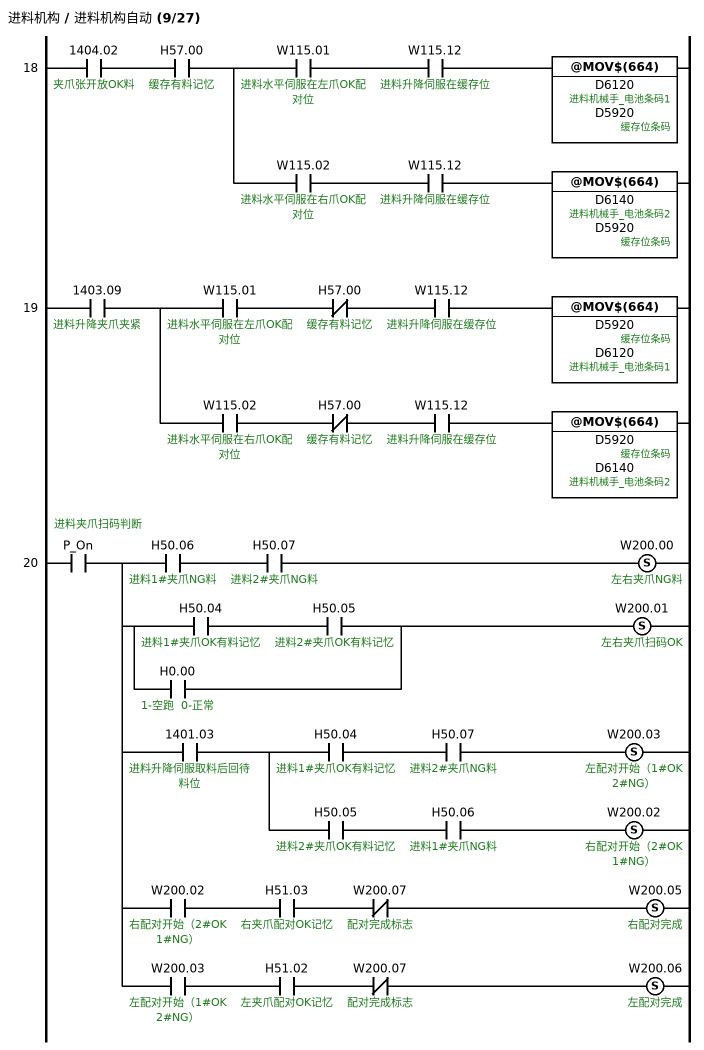
; rung 18
LD 1404.02  ; 夹爪张开放OK料
AND H57.00  ; 缓存有料记忆
OUT TR0
AND W115.01  ; 进料水平伺服在左爪OK配对位
AND W115.12  ; 进料升降伺服在缓存位
@MOV$(664) D6120 D5920  ; 进料机械手_电池条码1, 缓存位条码
LD TR0
AND W115.02  ; 进料水平伺服在右爪OK配对位
AND W115.12  ; 进料升降伺服在缓存位
@MOV$(664) D6140 D5920  ; 进料机械手_电池条码2, 缓存位条码
; rung 19
LD 1403.09  ; 进料升降夹爪夹紧
OUT TR0
AND W115.01  ; 进料水平伺服在左爪OK配对位
ANDNOT H57.00  ; 缓存有料记忆
AND W115.12  ; 进料升降伺服在缓存位
@MOV$(664) D5920 D6120  ; 缓存位条码, 进料机械手_电池条码1
LD TR0
AND W115.02  ; 进料水平伺服在右爪OK配对位
ANDNOT H57.00  ; 缓存有料记忆
AND W115.12  ; 进料升降伺服在缓存位
@MOV$(664) D5920 D6140  ; 缓存位条码, 进料机械手_电池条码2
; rung 20: 进料夹爪扫码判断
LD P_On
OUT TR0
AND H50.06  ; 进料1#夹爪NG料
AND H50.07  ; 进料2#夹爪NG料
SET W200.00  ; 左右夹爪NG料
LD TR0
LD H50.04  ; 进料1#夹爪OK有料记忆
AND H50.05  ; 进料2#夹爪OK有料记忆
OR H0.00  ; 1-空跑  0-正常
ANDLD
SET W200.01  ; 左右夹爪扫码OK
LD TR0
AND 1401.03  ; 进料升降伺服取料后回待料位
OUT TR1
AND H50.04  ; 进料1#夹爪OK有料记忆
AND H50.07  ; 进料2#夹爪NG料
SET W200.03  ; 左配对开始（1#OK 2#NG）
LD TR1
AND H50.05  ; 进料2#夹爪OK有料记忆
AND H50.06  ; 进料1#夹爪NG料
SET W200.02  ; 右配对开始（2#OK 1#NG）
LD TR0
AND W200.02  ; 右配对开始（2#OK 1#NG）
AND H51.03  ; 右夹爪配对OK记忆
ANDNOT W200.07  ; 配对完成标志
SET W200.05  ; 右配对完成
LD TR0
AND W200.03  ; 左配对开始（1#OK 2#NG）
AND H51.02  ; 左夹爪配对OK记忆
ANDNOT W200.07  ; 配对完成标志
SET W200.06  ; 左配对完成

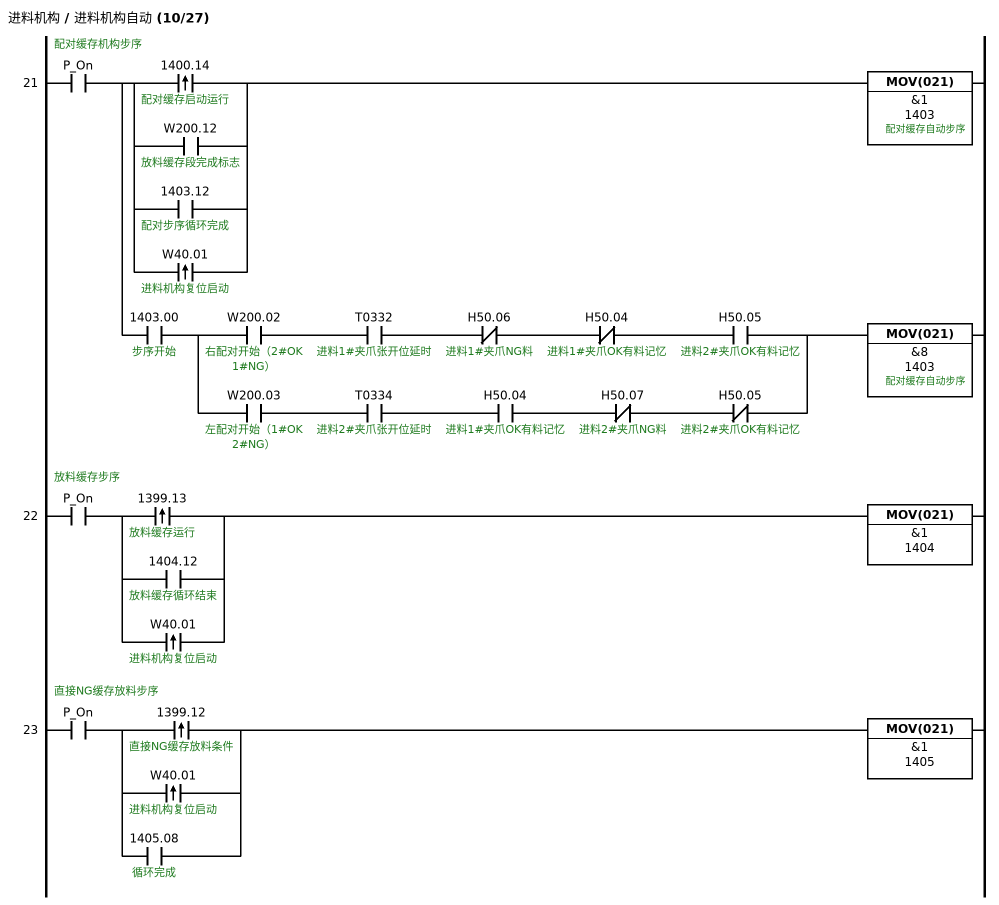
; rung 21: 配对缓存机构步序
LD P_On
OUT TR0
@LD 1400.14  ; 配对缓存启动运行
OR W200.12  ; 放料缓存段完成标志
OR 1403.12  ; 配对步序循环完成
@OR W40.01  ; 进料机构复位启动
ANDLD
MOV(021) &1 1403  ; 配对缓存自动步序
LD TR0
AND 1403.00  ; 步序开始
LD W200.02  ; 右配对开始（2#OK 1#NG）
AND T0332  ; 进料1#夹爪张开位延时
ANDNOT H50.06  ; 进料1#夹爪NG料
ANDNOT H50.04  ; 进料1#夹爪OK有料记忆
AND H50.05  ; 进料2#夹爪OK有料记忆
LD W200.03  ; 左配对开始（1#OK 2#NG）
AND T0334  ; 进料2#夹爪张开位延时
AND H50.04  ; 进料1#夹爪OK有料记忆
ANDNOT H50.07  ; 进料2#夹爪NG料
ANDNOT H50.05  ; 进料2#夹爪OK有料记忆
ORLD
ANDLD
MOV(021) &8 1403  ; 配对缓存自动步序
; rung 22: 放料缓存步序
LD P_On
@LD 1399.13  ; 放料缓存运行
OR 1404.12  ; 放料缓存循环结束
@OR W40.01  ; 进料机构复位启动
ANDLD
MOV(021) &1 1404
; rung 23: 直接NG缓存放料步序
LD P_On
@LD 1399.12  ; 直接NG缓存放料条件
@OR W40.01  ; 进料机构复位启动
OR 1405.08  ; 循环完成
ANDLD
MOV(021) &1 1405

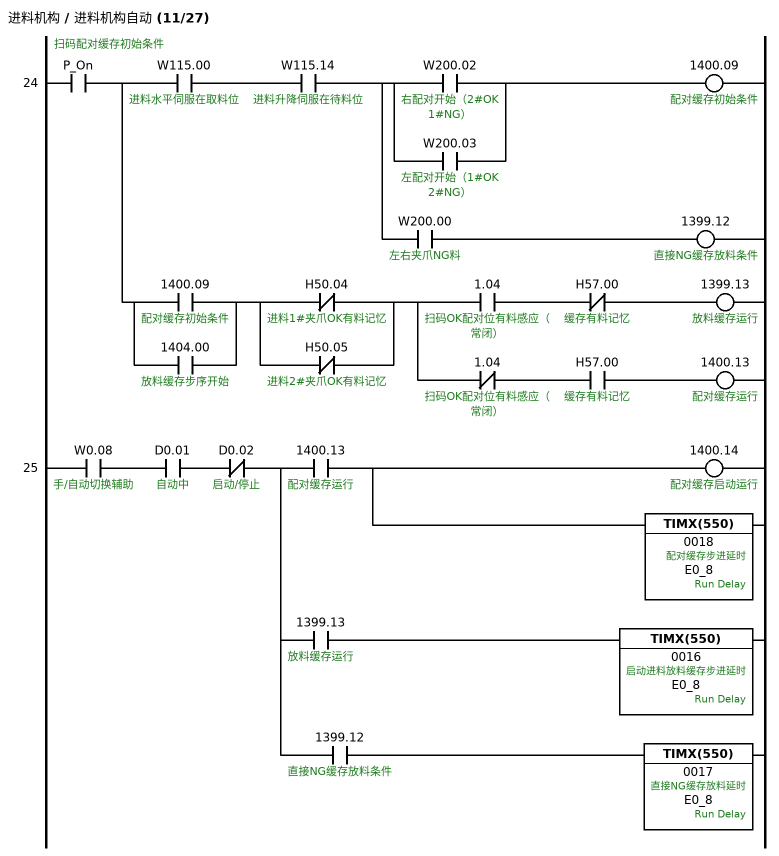
; rung 24: 扫码配对缓存初始条件
LD P_On
OUT TR0
AND W115.00  ; 进料水平伺服在取料位
AND W115.14  ; 进料升降伺服在待料位
OUT TR1
LD W200.02  ; 右配对开始（2#OK 1#NG）
OR W200.03  ; 左配对开始（1#OK 2#NG）
ANDLD
OUT 1400.09  ; 配对缓存初始条件
LD TR1
AND W200.00  ; 左右夹爪NG料
OUT 1399.12  ; 直接NG缓存放料条件
LD TR0
LD 1400.09  ; 配对缓存初始条件
OR 1404.00  ; 放料缓存步序开始
ANDLD
LDNOT H50.04  ; 进料1#夹爪OK有料记忆
ORNOT H50.05  ; 进料2#夹爪OK有料记忆
ANDLD
OUT TR0
AND 1.04  ; 扫码OK配对位有料感应（常闭）
ANDNOT H57.00  ; 缓存有料记忆
OUT 1399.13  ; 放料缓存运行
LD TR0
ANDNOT 1.04  ; 扫码OK配对位有料感应（常闭）
AND H57.00  ; 缓存有料记忆
OUT 1400.13  ; 配对缓存运行
; rung 25
LD W0.08  ; 手/自动切换辅助
AND D0.01  ; 自动中
ANDNOT D0.02  ; 启动/停止
OUT TR0
AND 1400.13  ; 配对缓存运行
OUT 1400.14  ; 配对缓存启动运行
TIMX(550) 0018 E0_8  ; Run Delay, 配对缓存步进延时
LD TR0
AND 1399.13  ; 放料缓存运行
TIMX(550) 0016 E0_8  ; Run Delay, 启动进料放料缓存步进延时
LD TR0
AND 1399.12  ; 直接NG缓存放料条件
TIMX(550) 0017 E0_8  ; Run Delay, 直接NG缓存放料延时

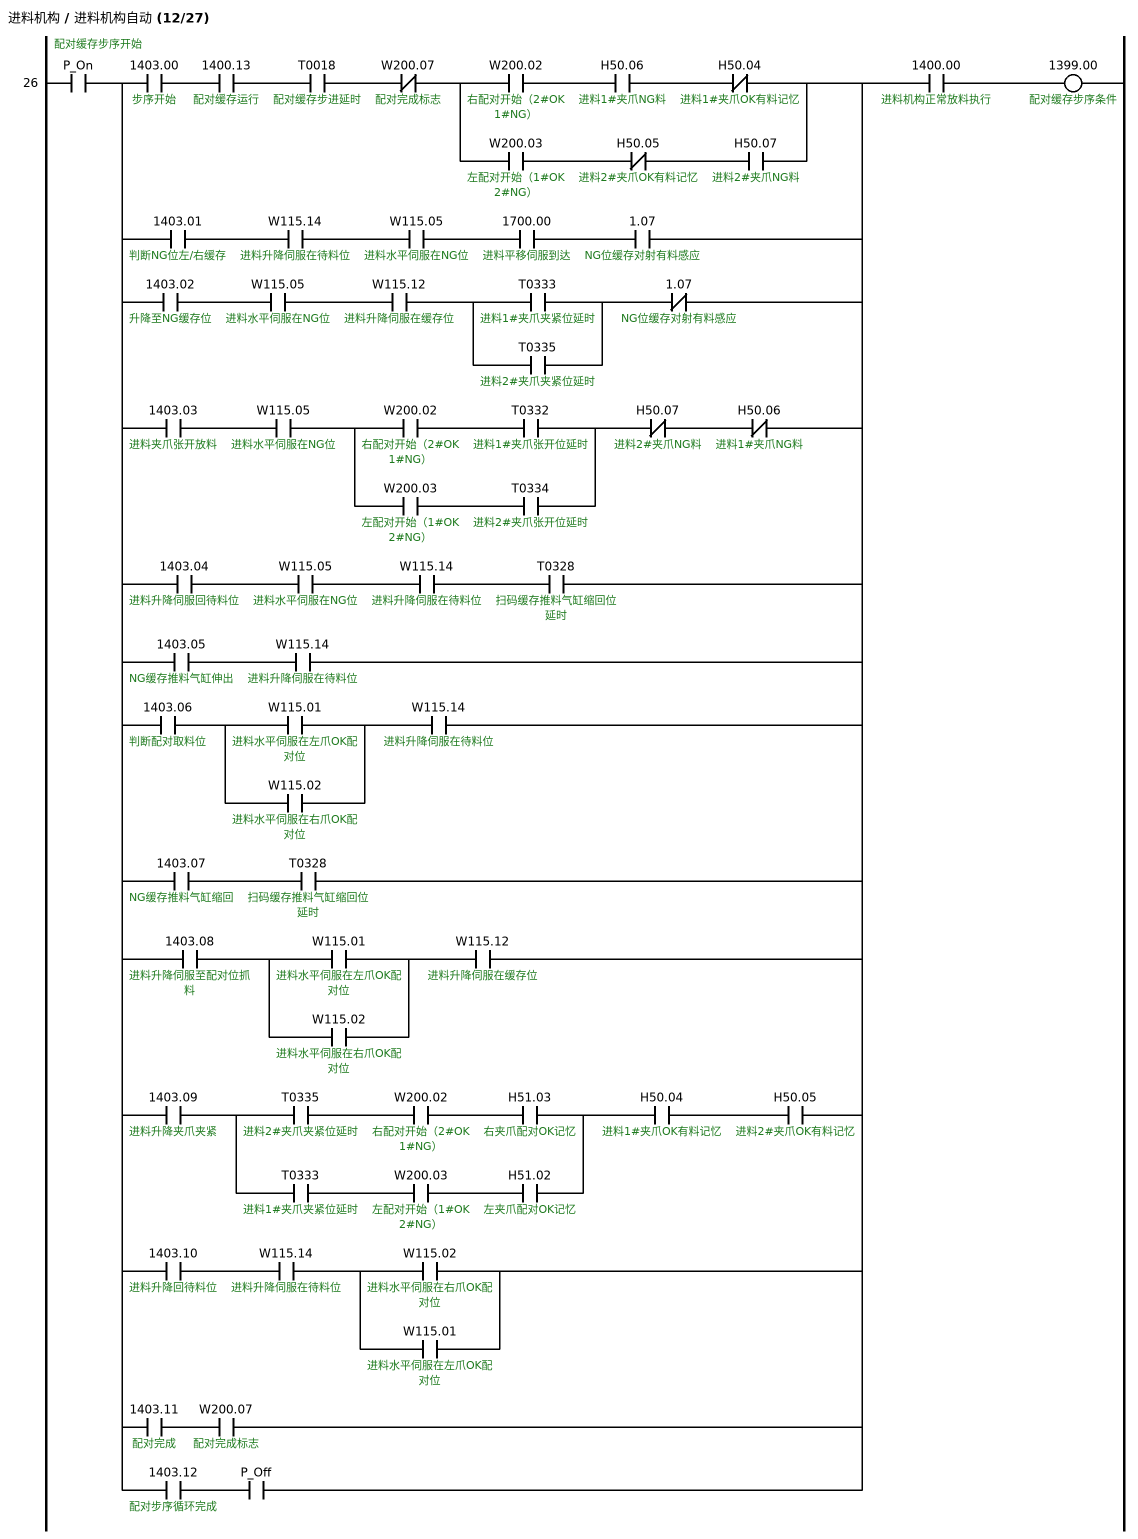
; rung 26: 配对缓存步序开始
LD P_On
LD 1403.00  ; 步序开始
AND 1400.13  ; 配对缓存运行
AND T0018  ; 配对缓存步进延时
ANDNOT W200.07  ; 配对完成标志
LD W200.02  ; 右配对开始（2#OK 1#NG）
AND H50.06  ; 进料1#夹爪NG料
ANDNOT H50.04  ; 进料1#夹爪OK有料记忆
LD W200.03  ; 左配对开始（1#OK 2#NG）
ANDNOT H50.05  ; 进料2#夹爪OK有料记忆
AND H50.07  ; 进料2#夹爪NG料
ORLD
ANDLD
LD 1403.01  ; 判断NG位左/右缓存
AND W115.14  ; 进料升降伺服在待料位
AND W115.05  ; 进料水平伺服在NG位
AND 1700.00  ; 进料平移伺服到达
AND 1.07  ; NG位缓存对射有料感应
ORLD
LD 1403.02  ; 升降至NG缓存位
AND W115.05  ; 进料水平伺服在NG位
AND W115.12  ; 进料升降伺服在缓存位
LD T0333  ; 进料1#夹爪夹紧位延时
OR T0335  ; 进料2#夹爪夹紧位延时
ANDLD
ANDNOT 1.07  ; NG位缓存对射有料感应
ORLD
LD 1403.03  ; 进料夹爪张开放料
AND W115.05  ; 进料水平伺服在NG位
LD W200.02  ; 右配对开始（2#OK 1#NG）
AND T0332  ; 进料1#夹爪张开位延时
LD W200.03  ; 左配对开始（1#OK 2#NG）
AND T0334  ; 进料2#夹爪张开位延时
ORLD
ANDLD
ANDNOT H50.07  ; 进料2#夹爪NG料
ANDNOT H50.06  ; 进料1#夹爪NG料
ORLD
LD 1403.04  ; 进料升降伺服回待料位
AND W115.05  ; 进料水平伺服在NG位
AND W115.14  ; 进料升降伺服在待料位
AND T0328  ; 扫码缓存推料气缸缩回位延时
ORLD
LD 1403.05  ; NG缓存推料气缸伸出
AND W115.14  ; 进料升降伺服在待料位
ORLD
LD 1403.06  ; 判断配对取料位
LD W115.01  ; 进料水平伺服在左爪OK配对位
OR W115.02  ; 进料水平伺服在右爪OK配对位
ANDLD
AND W115.14  ; 进料升降伺服在待料位
ORLD
LD 1403.07  ; NG缓存推料气缸缩回
AND T0328  ; 扫码缓存推料气缸缩回位延时
ORLD
LD 1403.08  ; 进料升降伺服至配对位抓料
LD W115.01  ; 进料水平伺服在左爪OK配对位
OR W115.02  ; 进料水平伺服在右爪OK配对位
ANDLD
AND W115.12  ; 进料升降伺服在缓存位
ORLD
LD 1403.09  ; 进料升降夹爪夹紧
LD T0335  ; 进料2#夹爪夹紧位延时
AND W200.02  ; 右配对开始（2#OK 1#NG）
AND H51.03  ; 右夹爪配对OK记忆
LD T0333  ; 进料1#夹爪夹紧位延时
AND W200.03  ; 左配对开始（1#OK 2#NG）
AND H51.02  ; 左夹爪配对OK记忆
ORLD
ANDLD
AND H50.04  ; 进料1#夹爪OK有料记忆
AND H50.05  ; 进料2#夹爪OK有料记忆
ORLD
LD 1403.10  ; 进料升降回待料位
AND W115.14  ; 进料升降伺服在待料位
LD W115.02  ; 进料水平伺服在右爪OK配对位
OR W115.01  ; 进料水平伺服在左爪OK配对位
ANDLD
ORLD
LD 1403.11  ; 配对完成
AND W200.07  ; 配对完成标志
ORLD
LD 1403.12  ; 配对步序循环完成
AND P_Off
ORLD
ANDLD
AND 1400.00  ; 进料机构正常放料执行
OUT 1399.00  ; 配对缓存步序条件

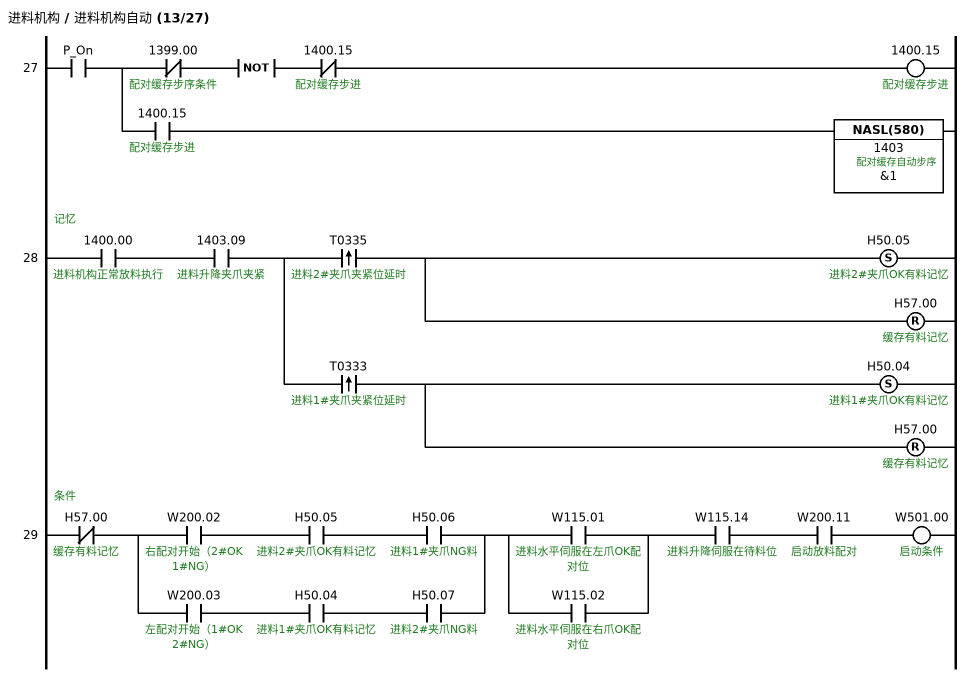
; rung 27
LD P_On
OUT TR0
ANDNOT 1399.00  ; 配对缓存步序条件
NOT(520)
ANDNOT 1400.15  ; 配对缓存步进
OUT 1400.15  ; 配对缓存步进
LD TR0
AND 1400.15  ; 配对缓存步进
NASL(580) 1403 &1  ; 配对缓存自动步序
; rung 28: 记忆
LD 1400.00  ; 进料机构正常放料执行
AND 1403.09  ; 进料升降夹爪夹紧
OUT TR0
@AND T0335  ; 进料2#夹爪夹紧位延时
SET H50.05  ; 进料2#夹爪OK有料记忆
RSET H57.00  ; 缓存有料记忆
LD TR0
@AND T0333  ; 进料1#夹爪夹紧位延时
SET H50.04  ; 进料1#夹爪OK有料记忆
RSET H57.00  ; 缓存有料记忆
; rung 29: 条件
LDNOT H57.00  ; 缓存有料记忆
LD W200.02  ; 右配对开始（2#OK 1#NG）
AND H50.05  ; 进料2#夹爪OK有料记忆
AND H50.06  ; 进料1#夹爪NG料
LD W200.03  ; 左配对开始（1#OK 2#NG）
AND H50.04  ; 进料1#夹爪OK有料记忆
AND H50.07  ; 进料2#夹爪NG料
ORLD
ANDLD
LD W115.01  ; 进料水平伺服在左爪OK配对位
OR W115.02  ; 进料水平伺服在右爪OK配对位
ANDLD
AND W115.14  ; 进料升降伺服在待料位
AND W200.11  ; 启动放料配对
OUT W501.00  ; 启动条件

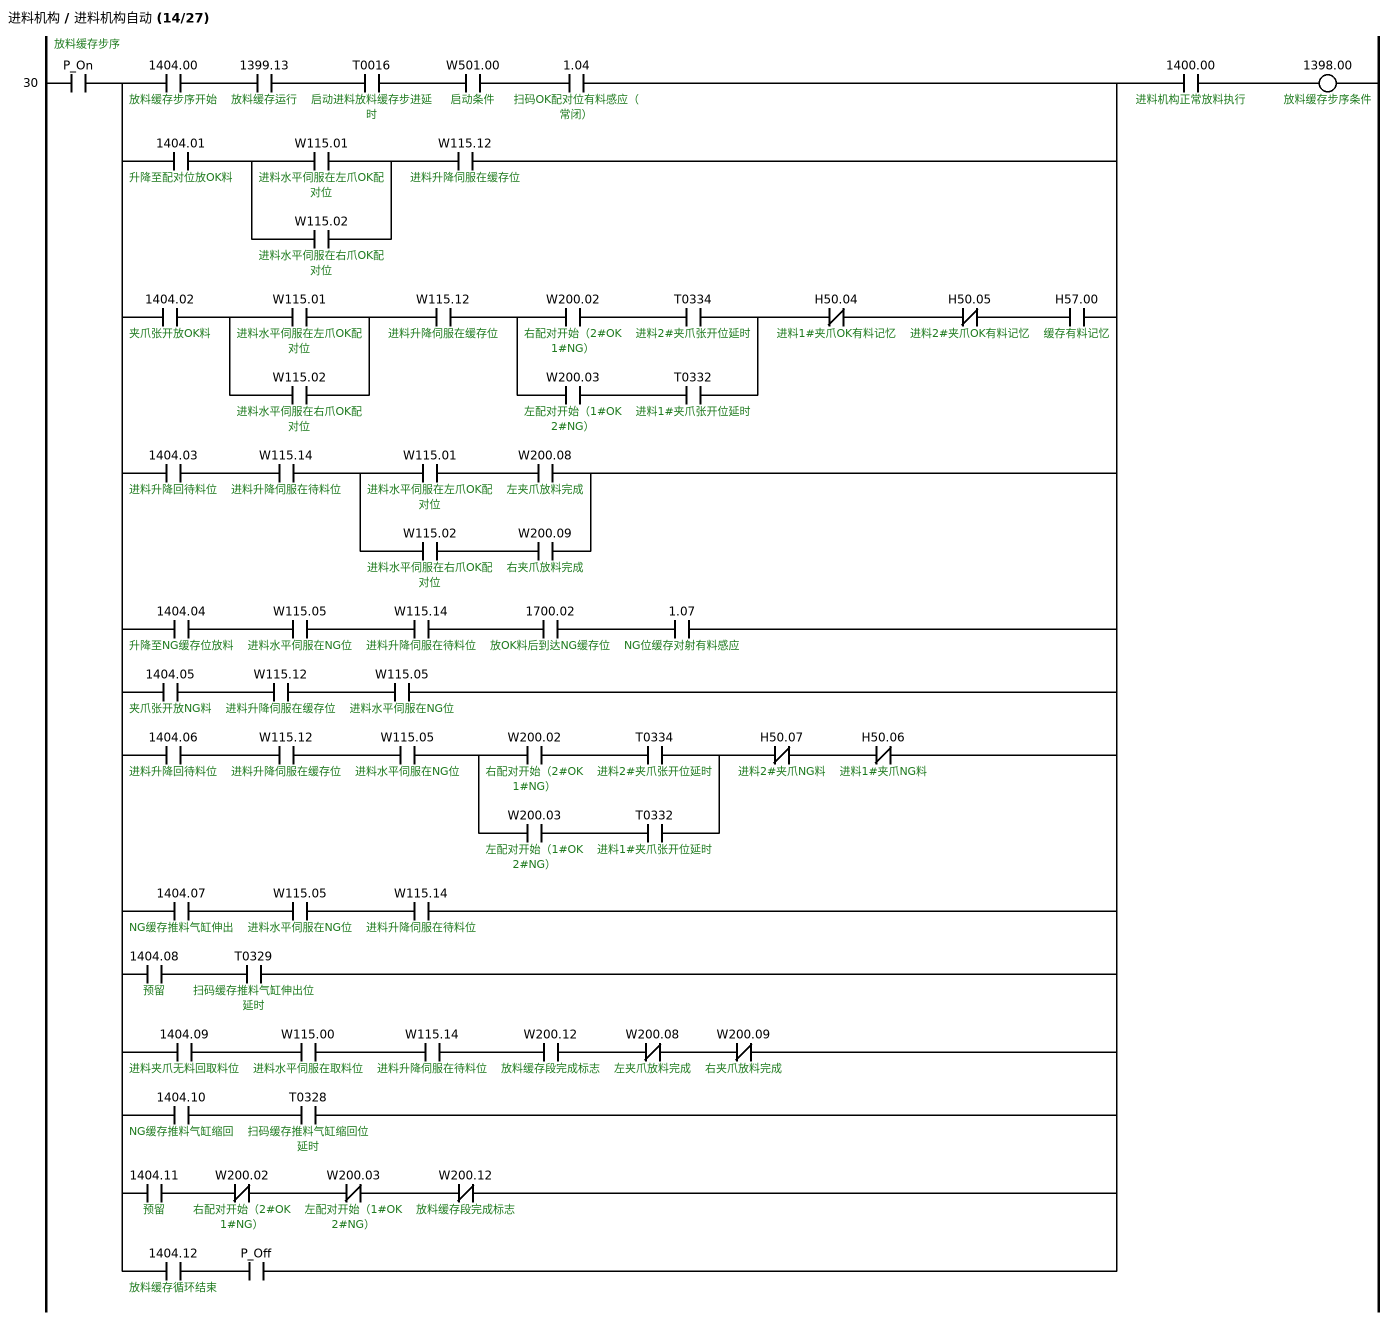
; rung 30: 放料缓存步序
LD P_On
LD 1404.00  ; 放料缓存步序开始
AND 1399.13  ; 放料缓存运行
AND T0016  ; 启动进料放料缓存步进延时
AND W501.00  ; 启动条件
AND 1.04  ; 扫码OK配对位有料感应（常闭）
LD 1404.01  ; 升降至配对位放OK料
LD W115.01  ; 进料水平伺服在左爪OK配对位
OR W115.02  ; 进料水平伺服在右爪OK配对位
ANDLD
AND W115.12  ; 进料升降伺服在缓存位
ORLD
LD 1404.02  ; 夹爪张开放OK料
LD W115.01  ; 进料水平伺服在左爪OK配对位
OR W115.02  ; 进料水平伺服在右爪OK配对位
ANDLD
AND W115.12  ; 进料升降伺服在缓存位
LD W200.02  ; 右配对开始（2#OK 1#NG）
AND T0334  ; 进料2#夹爪张开位延时
LD W200.03  ; 左配对开始（1#OK 2#NG）
AND T0332  ; 进料1#夹爪张开位延时
ORLD
ANDLD
ANDNOT H50.04  ; 进料1#夹爪OK有料记忆
ANDNOT H50.05  ; 进料2#夹爪OK有料记忆
AND H57.00  ; 缓存有料记忆
ORLD
LD 1404.03  ; 进料升降回待料位
AND W115.14  ; 进料升降伺服在待料位
LD W115.01  ; 进料水平伺服在左爪OK配对位
AND W200.08  ; 左夹爪放料完成
LD W115.02  ; 进料水平伺服在右爪OK配对位
AND W200.09  ; 右夹爪放料完成
ORLD
ANDLD
ORLD
LD 1404.04  ; 升降至NG缓存位放料
AND W115.05  ; 进料水平伺服在NG位
AND W115.14  ; 进料升降伺服在待料位
AND 1700.02  ; 放OK料后到达NG缓存位
AND 1.07  ; NG位缓存对射有料感应
ORLD
LD 1404.05  ; 夹爪张开放NG料
AND W115.12  ; 进料升降伺服在缓存位
AND W115.05  ; 进料水平伺服在NG位
ORLD
LD 1404.06  ; 进料升降回待料位
AND W115.12  ; 进料升降伺服在缓存位
AND W115.05  ; 进料水平伺服在NG位
LD W200.02  ; 右配对开始（2#OK 1#NG）
AND T0334  ; 进料2#夹爪张开位延时
LD W200.03  ; 左配对开始（1#OK 2#NG）
AND T0332  ; 进料1#夹爪张开位延时
ORLD
ANDLD
ANDNOT H50.07  ; 进料2#夹爪NG料
ANDNOT H50.06  ; 进料1#夹爪NG料
ORLD
LD 1404.07  ; NG缓存推料气缸伸出
AND W115.05  ; 进料水平伺服在NG位
AND W115.14  ; 进料升降伺服在待料位
ORLD
LD 1404.08  ; 预留
AND T0329  ; 扫码缓存推料气缸伸出位延时
ORLD
LD 1404.09  ; 进料夹爪无料回取料位
AND W115.00  ; 进料水平伺服在取料位
AND W115.14  ; 进料升降伺服在待料位
AND W200.12  ; 放料缓存段完成标志
ANDNOT W200.08  ; 左夹爪放料完成
ANDNOT W200.09  ; 右夹爪放料完成
ORLD
LD 1404.10  ; NG缓存推料气缸缩回
AND T0328  ; 扫码缓存推料气缸缩回位延时
ORLD
LD 1404.11  ; 预留
ANDNOT W200.02  ; 右配对开始（2#OK 1#NG）
ANDNOT W200.03  ; 左配对开始（1#OK 2#NG）
ANDNOT W200.12  ; 放料缓存段完成标志
ORLD
LD 1404.12  ; 放料缓存循环结束
AND P_Off
ORLD
ANDLD
AND 1400.00  ; 进料机构正常放料执行
OUT 1398.00  ; 放料缓存步序条件

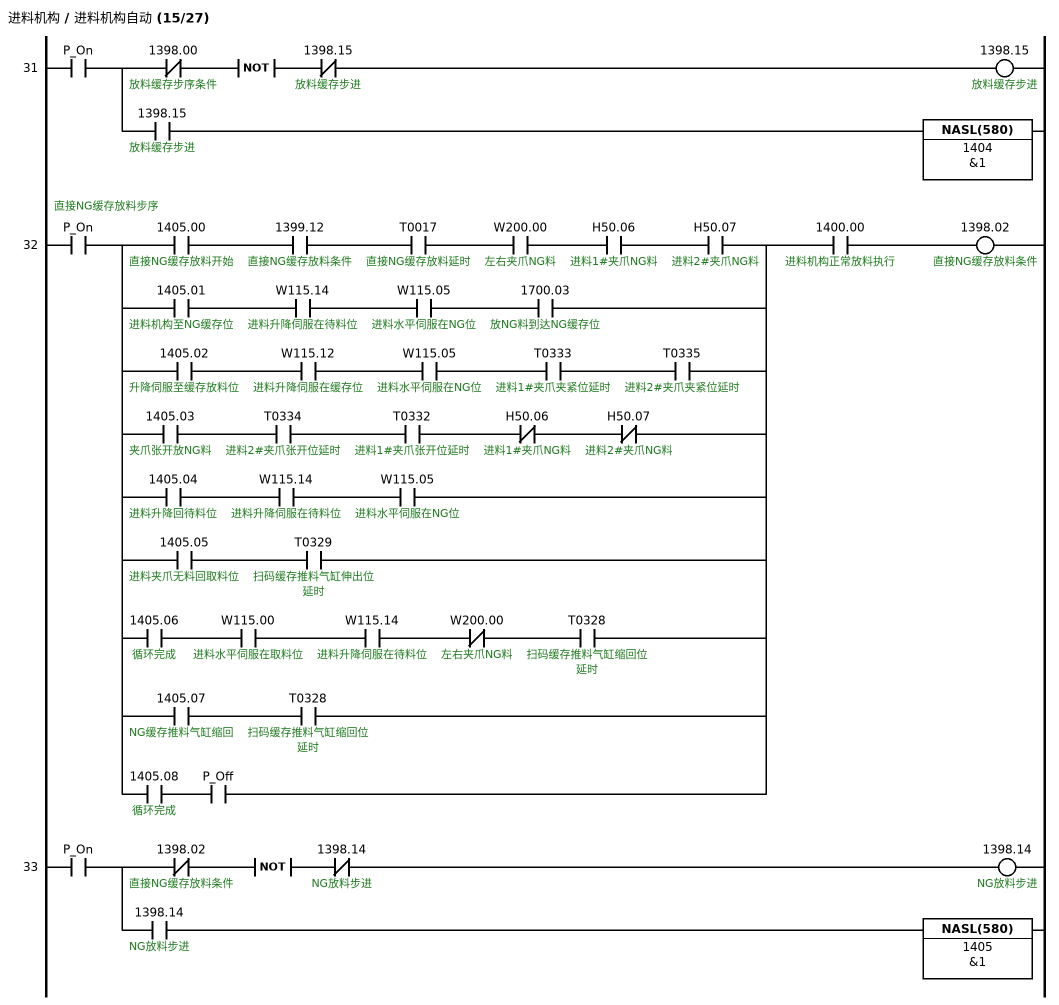
; rung 31
LD P_On
OUT TR0
ANDNOT 1398.00  ; 放料缓存步序条件
NOT(520)
ANDNOT 1398.15  ; 放料缓存步进
OUT 1398.15  ; 放料缓存步进
LD TR0
AND 1398.15  ; 放料缓存步进
NASL(580) 1404 &1
; rung 32: 直接NG缓存放料步序
LD P_On
LD 1405.00  ; 直接NG缓存放料开始
AND 1399.12  ; 直接NG缓存放料条件
AND T0017  ; 直接NG缓存放料延时
AND W200.00  ; 左右夹爪NG料
AND H50.06  ; 进料1#夹爪NG料
AND H50.07  ; 进料2#夹爪NG料
LD 1405.01  ; 进料机构至NG缓存位
AND W115.14  ; 进料升降伺服在待料位
AND W115.05  ; 进料水平伺服在NG位
AND 1700.03  ; 放NG料到达NG缓存位
ORLD
LD 1405.02  ; 升降伺服至缓存放料位
AND W115.12  ; 进料升降伺服在缓存位
AND W115.05  ; 进料水平伺服在NG位
AND T0333  ; 进料1#夹爪夹紧位延时
AND T0335  ; 进料2#夹爪夹紧位延时
ORLD
LD 1405.03  ; 夹爪张开放NG料
AND T0334  ; 进料2#夹爪张开位延时
AND T0332  ; 进料1#夹爪张开位延时
ANDNOT H50.06  ; 进料1#夹爪NG料
ANDNOT H50.07  ; 进料2#夹爪NG料
ORLD
LD 1405.04  ; 进料升降回待料位
AND W115.14  ; 进料升降伺服在待料位
AND W115.05  ; 进料水平伺服在NG位
ORLD
LD 1405.05  ; 进料夹爪无料回取料位
AND T0329  ; 扫码缓存推料气缸伸出位延时
ORLD
LD 1405.06  ; 循环完成
AND W115.00  ; 进料水平伺服在取料位
AND W115.14  ; 进料升降伺服在待料位
ANDNOT W200.00  ; 左右夹爪NG料
AND T0328  ; 扫码缓存推料气缸缩回位延时
ORLD
LD 1405.07  ; NG缓存推料气缸缩回
AND T0328  ; 扫码缓存推料气缸缩回位延时
ORLD
LD 1405.08  ; 循环完成
AND P_Off
ORLD
ANDLD
AND 1400.00  ; 进料机构正常放料执行
OUT 1398.02  ; 直接NG缓存放料条件
; rung 33
LD P_On
OUT TR0
ANDNOT 1398.02  ; 直接NG缓存放料条件
NOT(520)
ANDNOT 1398.14  ; NG放料步进
OUT 1398.14  ; NG放料步进
LD TR0
AND 1398.14  ; NG放料步进
NASL(580) 1405 &1

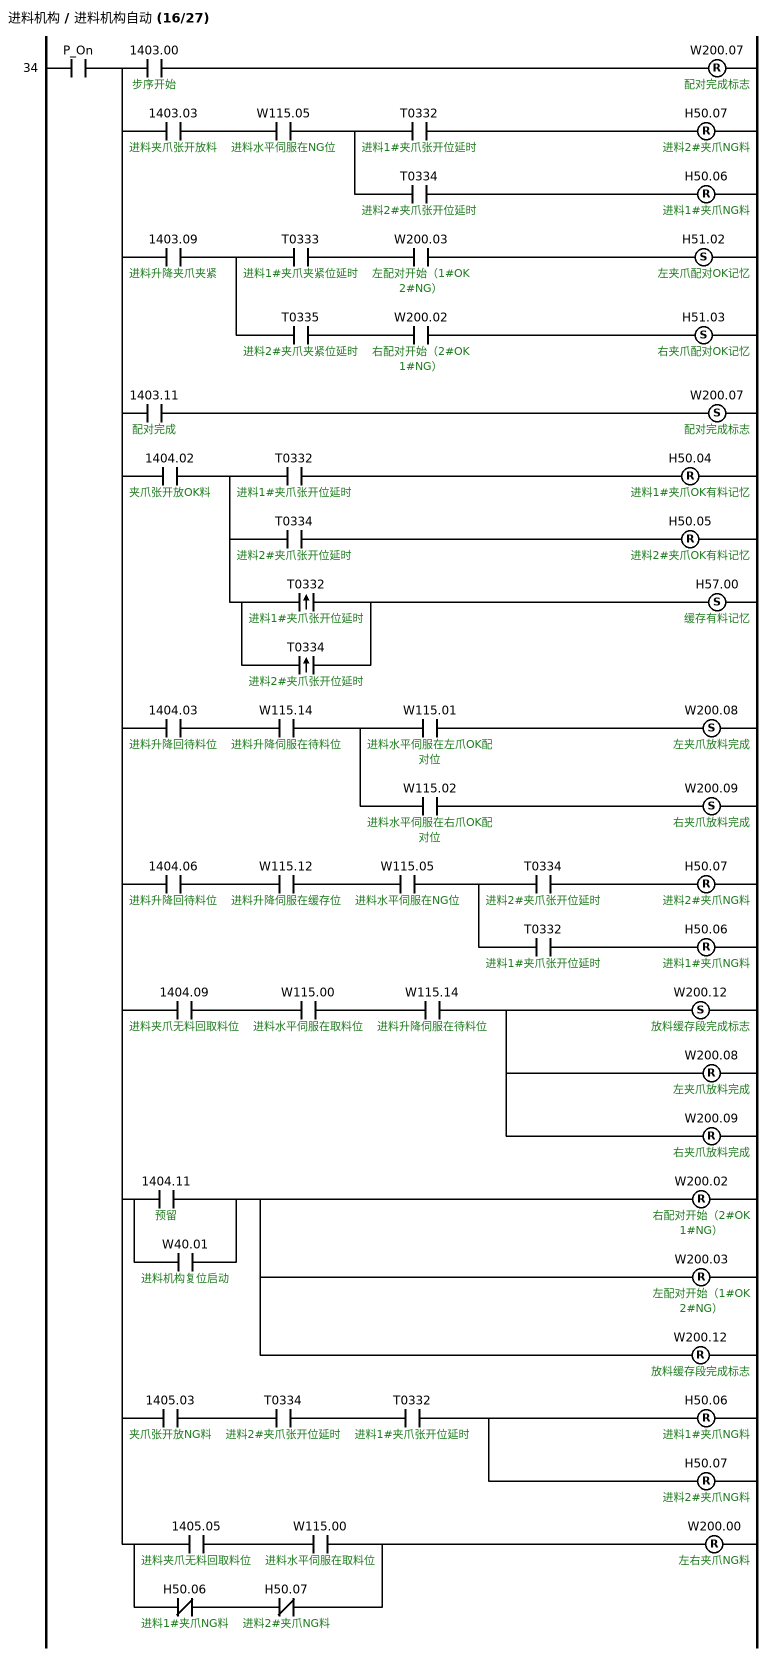
; rung 34
LD P_On
OUT TR0
AND 1403.00  ; 步序开始
RSET W200.07  ; 配对完成标志
LD TR0
AND 1403.03  ; 进料夹爪张开放料
AND W115.05  ; 进料水平伺服在NG位
OUT TR1
AND T0332  ; 进料1#夹爪张开位延时
RSET H50.07  ; 进料2#夹爪NG料
LD TR1
AND T0334  ; 进料2#夹爪张开位延时
RSET H50.06  ; 进料1#夹爪NG料
LD TR0
AND 1403.09  ; 进料升降夹爪夹紧
OUT TR1
AND T0333  ; 进料1#夹爪夹紧位延时
AND W200.03  ; 左配对开始（1#OK 2#NG）
SET H51.02  ; 左夹爪配对OK记忆
LD TR1
AND T0335  ; 进料2#夹爪夹紧位延时
AND W200.02  ; 右配对开始（2#OK 1#NG）
SET H51.03  ; 右夹爪配对OK记忆
LD TR0
AND 1403.11  ; 配对完成
SET W200.07  ; 配对完成标志
LD TR0
AND 1404.02  ; 夹爪张开放OK料
OUT TR1
AND T0332  ; 进料1#夹爪张开位延时
RSET H50.04  ; 进料1#夹爪OK有料记忆
LD TR1
AND T0334  ; 进料2#夹爪张开位延时
RSET H50.05  ; 进料2#夹爪OK有料记忆
LD TR1
@LD T0332  ; 进料1#夹爪张开位延时
@OR T0334  ; 进料2#夹爪张开位延时
ANDLD
SET H57.00  ; 缓存有料记忆
LD TR0
AND 1404.03  ; 进料升降回待料位
AND W115.14  ; 进料升降伺服在待料位
OUT TR1
AND W115.01  ; 进料水平伺服在左爪OK配对位
SET W200.08  ; 左夹爪放料完成
LD TR1
AND W115.02  ; 进料水平伺服在右爪OK配对位
SET W200.09  ; 右夹爪放料完成
LD TR0
AND 1404.06  ; 进料升降回待料位
AND W115.12  ; 进料升降伺服在缓存位
AND W115.05  ; 进料水平伺服在NG位
OUT TR1
AND T0334  ; 进料2#夹爪张开位延时
RSET H50.07  ; 进料2#夹爪NG料
LD TR1
AND T0332  ; 进料1#夹爪张开位延时
RSET H50.06  ; 进料1#夹爪NG料
LD TR0
AND 1404.09  ; 进料夹爪无料回取料位
AND W115.00  ; 进料水平伺服在取料位
AND W115.14  ; 进料升降伺服在待料位
SET W200.12  ; 放料缓存段完成标志
RSET W200.08  ; 左夹爪放料完成
RSET W200.09  ; 右夹爪放料完成
LD TR0
LD 1404.11  ; 预留
OR W40.01  ; 进料机构复位启动
ANDLD
RSET W200.02  ; 右配对开始（2#OK 1#NG）
RSET W200.03  ; 左配对开始（1#OK 2#NG）
RSET W200.12  ; 放料缓存段完成标志
LD TR0
AND 1405.03  ; 夹爪张开放NG料
AND T0334  ; 进料2#夹爪张开位延时
AND T0332  ; 进料1#夹爪张开位延时
RSET H50.06  ; 进料1#夹爪NG料
RSET H50.07  ; 进料2#夹爪NG料
LD TR0
LD 1405.05  ; 进料夹爪无料回取料位
AND W115.00  ; 进料水平伺服在取料位
LDNOT H50.06  ; 进料1#夹爪NG料
ANDNOT H50.07  ; 进料2#夹爪NG料
ORLD
ANDLD
RSET W200.00  ; 左右夹爪NG料

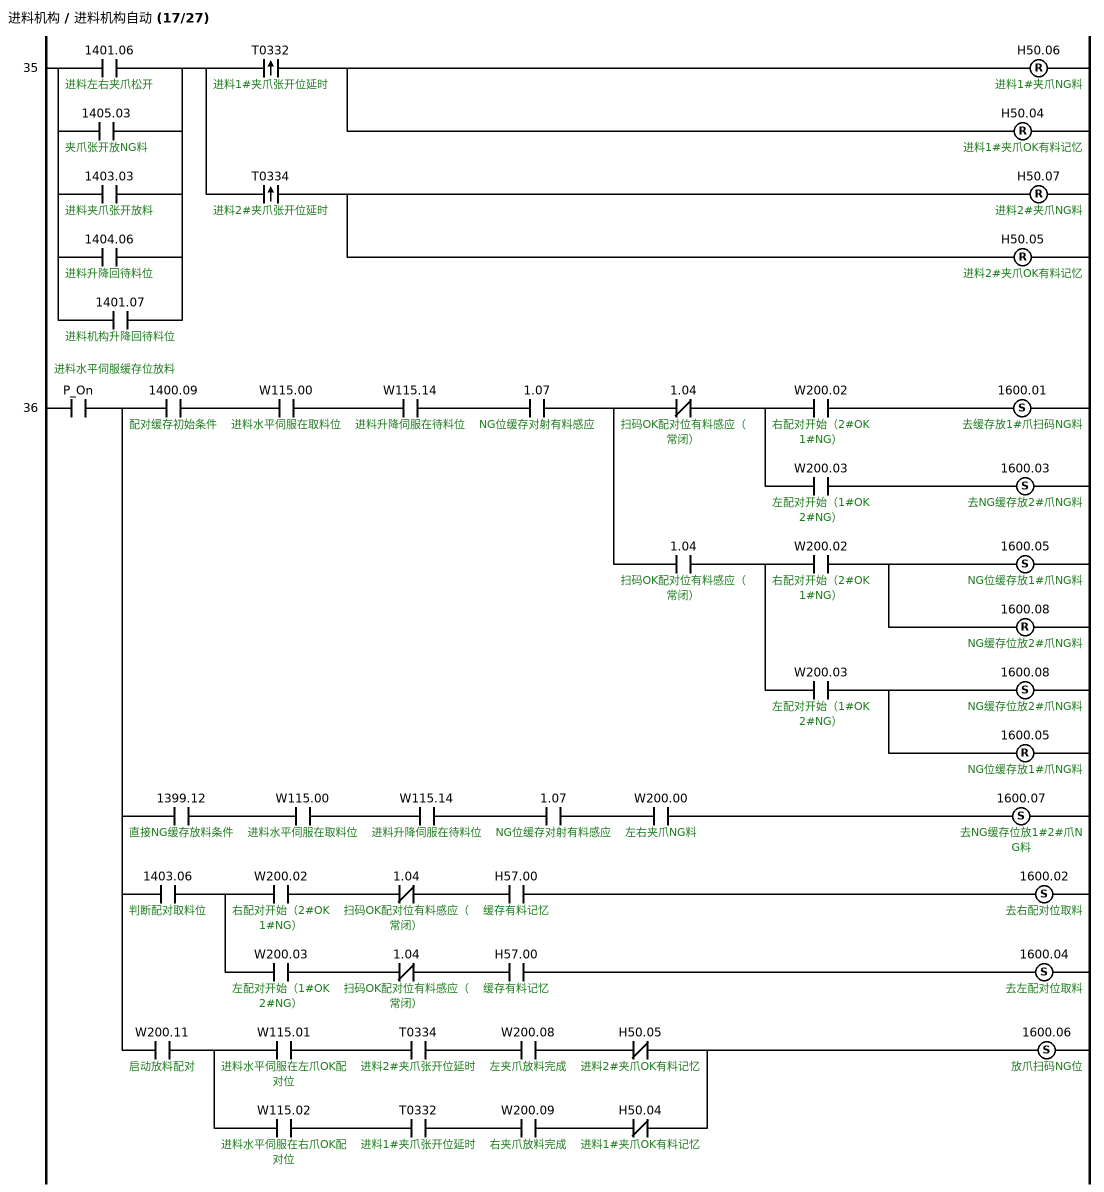
; rung 35
LD 1401.06  ; 进料左右夹爪松开
OR 1405.03  ; 夹爪张开放NG料
OR 1403.03  ; 进料夹爪张开放料
OR 1404.06  ; 进料升降回待料位
OR 1401.07  ; 进料机构升降回待料位
OUT TR0
@AND T0332  ; 进料1#夹爪张开位延时
RSET H50.06  ; 进料1#夹爪NG料
RSET H50.04  ; 进料1#夹爪OK有料记忆
LD TR0
@AND T0334  ; 进料2#夹爪张开位延时
RSET H50.07  ; 进料2#夹爪NG料
RSET H50.05  ; 进料2#夹爪OK有料记忆
; rung 36: 进料水平伺服缓存位放料
LD P_On
OUT TR0
AND 1400.09  ; 配对缓存初始条件
AND W115.00  ; 进料水平伺服在取料位
AND W115.14  ; 进料升降伺服在待料位
AND 1.07  ; NG位缓存对射有料感应
OUT TR1
ANDNOT 1.04  ; 扫码OK配对位有料感应（常闭）
OUT TR2
AND W200.02  ; 右配对开始（2#OK 1#NG）
SET 1600.01  ; 去缓存放1#爪扫码NG料
LD TR2
AND W200.03  ; 左配对开始（1#OK 2#NG）
SET 1600.03  ; 去NG缓存放2#爪NG料
LD TR1
AND 1.04  ; 扫码OK配对位有料感应（常闭）
OUT TR1
AND W200.02  ; 右配对开始（2#OK 1#NG）
SET 1600.05  ; NG位缓存放1#爪NG料
RSET 1600.08  ; NG缓存位放2#爪NG料
LD TR1
AND W200.03  ; 左配对开始（1#OK 2#NG）
SET 1600.08  ; NG缓存位放2#爪NG料
RSET 1600.05  ; NG位缓存放1#爪NG料
LD TR0
AND 1399.12  ; 直接NG缓存放料条件
AND W115.00  ; 进料水平伺服在取料位
AND W115.14  ; 进料升降伺服在待料位
AND 1.07  ; NG位缓存对射有料感应
AND W200.00  ; 左右夹爪NG料
SET 1600.07  ; 去NG缓存位放1#2#爪NG料
LD TR0
AND 1403.06  ; 判断配对取料位
OUT TR1
AND W200.02  ; 右配对开始（2#OK 1#NG）
ANDNOT 1.04  ; 扫码OK配对位有料感应（常闭）
AND H57.00  ; 缓存有料记忆
SET 1600.02  ; 去右配对位取料
LD TR1
AND W200.03  ; 左配对开始（1#OK 2#NG）
ANDNOT 1.04  ; 扫码OK配对位有料感应（常闭）
AND H57.00  ; 缓存有料记忆
SET 1600.04  ; 去左配对位取料
LD TR0
AND W200.11  ; 启动放料配对
LD W115.01  ; 进料水平伺服在左爪OK配对位
AND T0334  ; 进料2#夹爪张开位延时
AND W200.08  ; 左夹爪放料完成
ANDNOT H50.05  ; 进料2#夹爪OK有料记忆
LD W115.02  ; 进料水平伺服在右爪OK配对位
AND T0332  ; 进料1#夹爪张开位延时
AND W200.09  ; 右夹爪放料完成
ANDNOT H50.04  ; 进料1#夹爪OK有料记忆
ORLD
ANDLD
SET 1600.06  ; 放爪扫码NG位

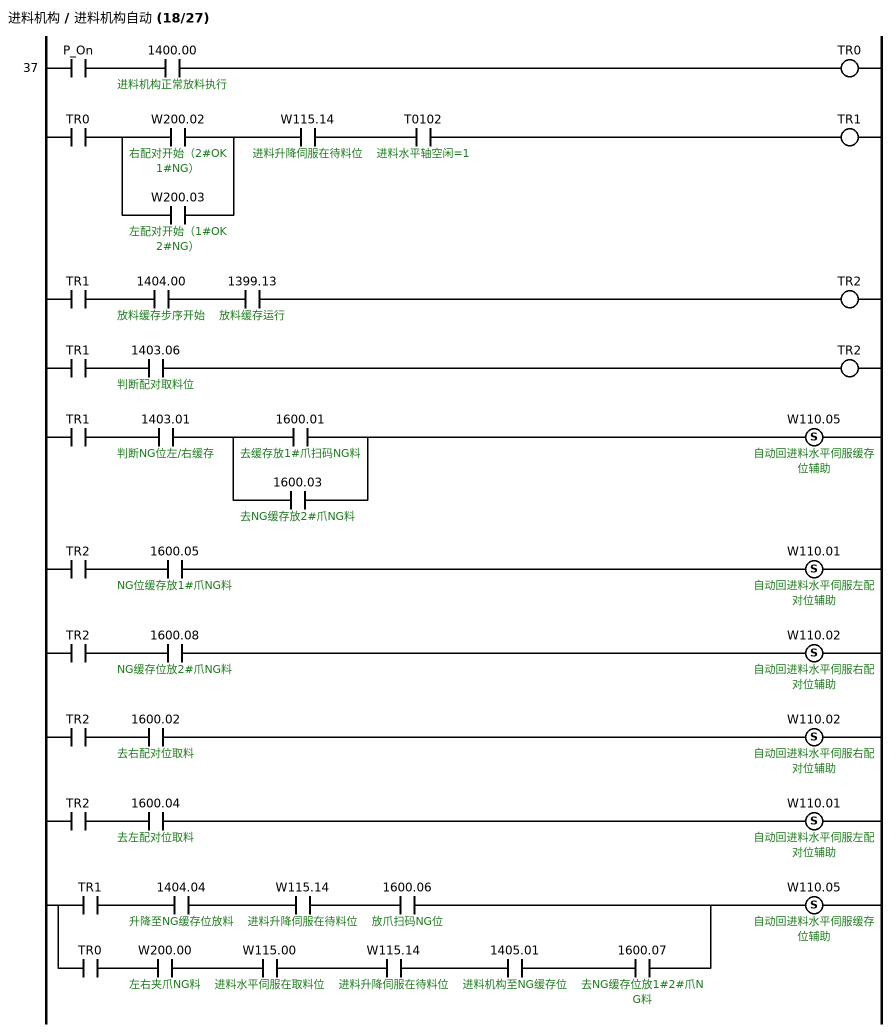
; rung 37
LD P_On
AND 1400.00  ; 进料机构正常放料执行
OUT TR0
LD W200.02  ; 右配对开始（2#OK 1#NG）
OR W200.03  ; 左配对开始（1#OK 2#NG）
ANDLD
AND W115.14  ; 进料升降伺服在待料位
AND T0102  ; 进料水平轴空闲=1
OUT TR1
AND 1403.01  ; 判断NG位左/右缓存
LD 1600.01  ; 去缓存放1#爪扫码NG料
OR 1600.03  ; 去NG缓存放2#爪NG料
ANDLD
SET W110.05  ; 自动回进料水平伺服缓存位辅助
LD TR1
AND 1404.00  ; 放料缓存步序开始
AND 1399.13  ; 放料缓存运行
OUT TR2
AND 1600.05  ; NG位缓存放1#爪NG料
SET W110.01  ; 自动回进料水平伺服左配对位辅助
LD TR2
AND 1600.08  ; NG缓存位放2#爪NG料
SET W110.02  ; 自动回进料水平伺服右配对位辅助
LD TR1
AND 1403.06  ; 判断配对取料位
OUT TR2
AND 1600.02  ; 去右配对位取料
SET W110.02  ; 自动回进料水平伺服右配对位辅助
LD TR2
AND 1600.04  ; 去左配对位取料
SET W110.01  ; 自动回进料水平伺服左配对位辅助
LD TR1
AND 1404.04  ; 升降至NG缓存位放料
AND W115.14  ; 进料升降伺服在待料位
AND 1600.06  ; 放爪扫码NG位
LD TR0
AND W200.00  ; 左右夹爪NG料
AND W115.00  ; 进料水平伺服在取料位
AND W115.14  ; 进料升降伺服在待料位
AND 1405.01  ; 进料机构至NG缓存位
AND 1600.07  ; 去NG缓存位放1#2#爪NG料
ORLD
SET W110.05  ; 自动回进料水平伺服缓存位辅助

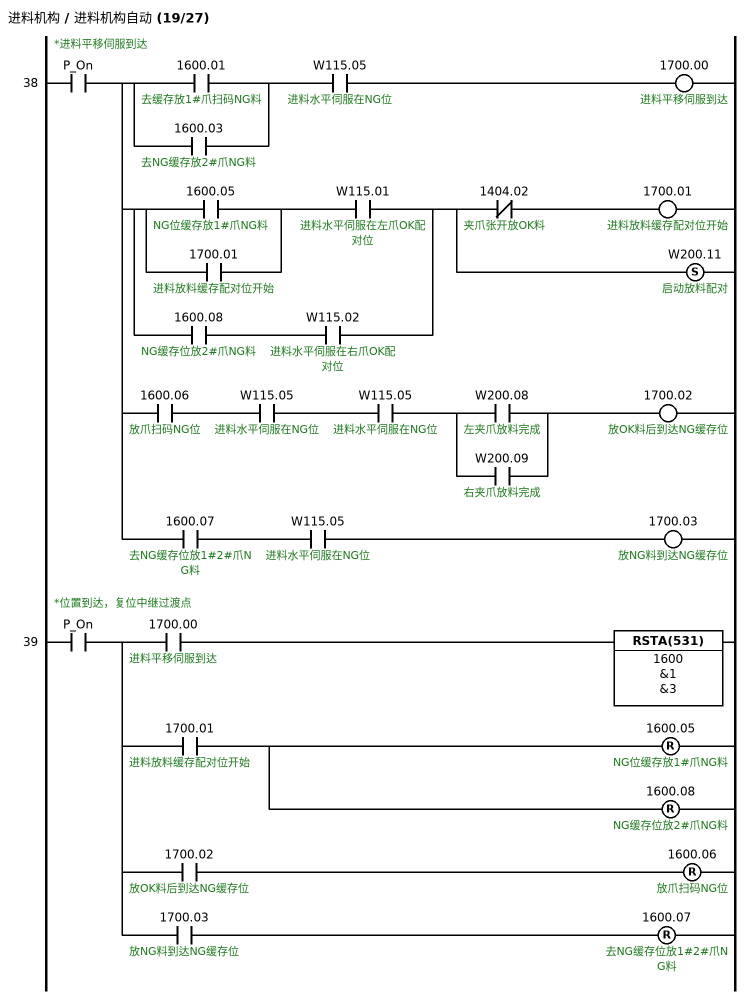
; rung 38: *进料平移伺服到达
LD P_On
OUT TR0
LD 1600.01  ; 去缓存放1#爪扫码NG料
OR 1600.03  ; 去NG缓存放2#爪NG料
ANDLD
AND W115.05  ; 进料水平伺服在NG位
OUT 1700.00  ; 进料平移伺服到达
LD TR0
LD 1600.05  ; NG位缓存放1#爪NG料
OR 1700.01  ; 进料放料缓存配对位开始
AND W115.01  ; 进料水平伺服在左爪OK配对位
LD 1600.08  ; NG缓存位放2#爪NG料
AND W115.02  ; 进料水平伺服在右爪OK配对位
ORLD
ANDLD
OUT TR1
ANDNOT 1404.02  ; 夹爪张开放OK料
OUT 1700.01  ; 进料放料缓存配对位开始
LD TR1
SET W200.11  ; 启动放料配对
LD TR0
AND 1600.06  ; 放爪扫码NG位
AND W115.05  ; 进料水平伺服在NG位
AND W115.05  ; 进料水平伺服在NG位
LD W200.08  ; 左夹爪放料完成
OR W200.09  ; 右夹爪放料完成
ANDLD
OUT 1700.02  ; 放OK料后到达NG缓存位
LD TR0
AND 1600.07  ; 去NG缓存位放1#2#爪NG料
AND W115.05  ; 进料水平伺服在NG位
OUT 1700.03  ; 放NG料到达NG缓存位
; rung 39: *位置到达，复位中继过渡点
LD P_On
OUT TR0
AND 1700.00  ; 进料平移伺服到达
RSTA(531) 1600 &1 &3
LD TR0
AND 1700.01  ; 进料放料缓存配对位开始
RSET 1600.05  ; NG位缓存放1#爪NG料
RSET 1600.08  ; NG缓存位放2#爪NG料
LD TR0
AND 1700.02  ; 放OK料后到达NG缓存位
RSET 1600.06  ; 放爪扫码NG位
LD TR0
AND 1700.03  ; 放NG料到达NG缓存位
RSET 1600.07  ; 去NG缓存位放1#2#爪NG料

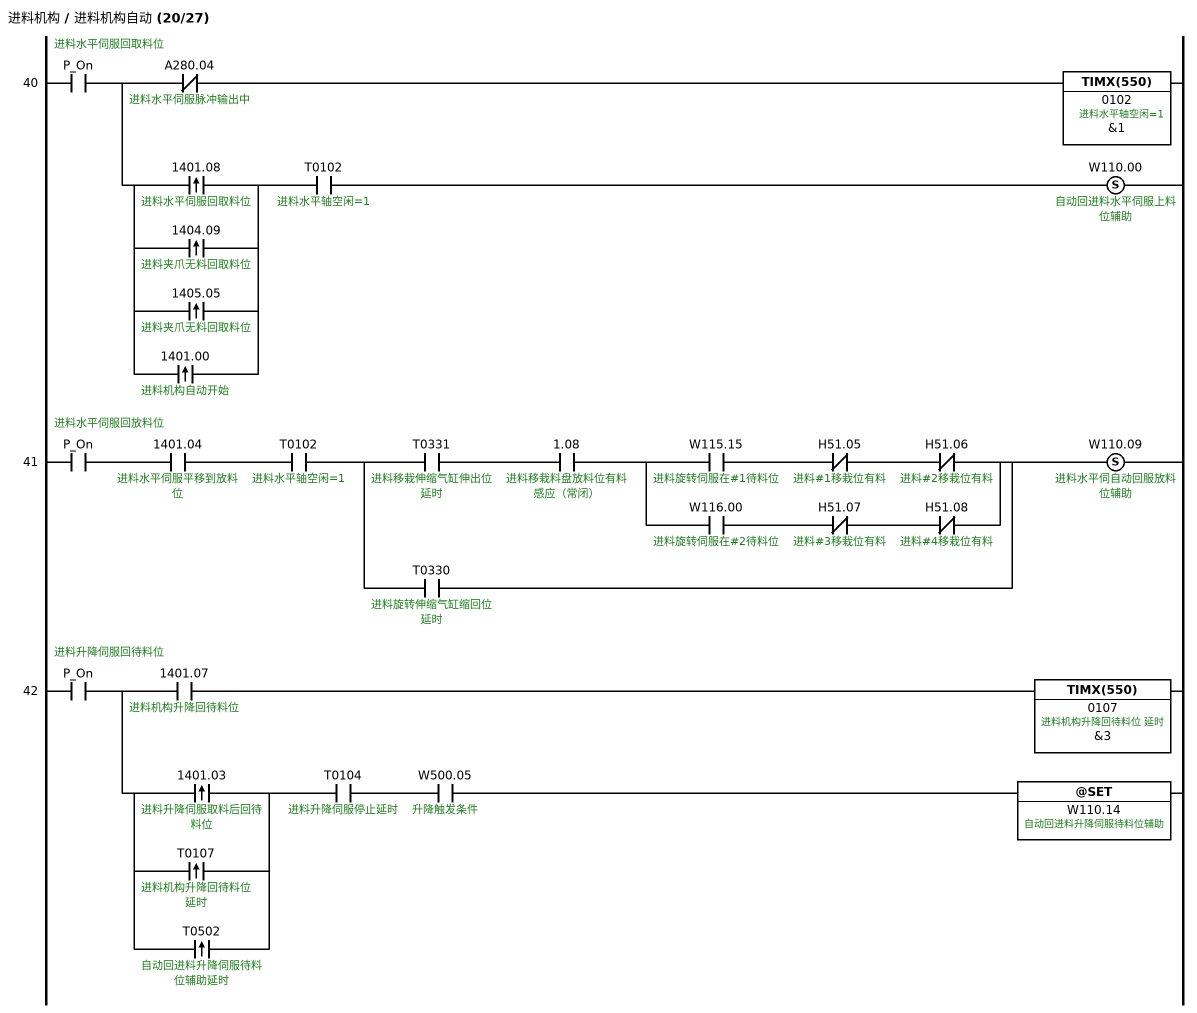
; rung 40: 进料水平伺服回取料位
LD P_On
OUT TR0
ANDNOT A280.04  ; 进料水平伺服脉冲输出中
TIMX(550) 0102 &1  ; 进料水平轴空闲=1
LD TR0
@LD 1401.08  ; 进料水平伺服回取料位
@OR 1404.09  ; 进料夹爪无料回取料位
@OR 1405.05  ; 进料夹爪无料回取料位
@OR 1401.00  ; 进料机构自动开始
ANDLD
AND T0102  ; 进料水平轴空闲=1
SET W110.00  ; 自动回进料水平伺服上料位辅助
; rung 41: 进料水平伺服回放料位
LD P_On
AND 1401.04  ; 进料水平伺服平移到放料位
AND T0102  ; 进料水平轴空闲=1
LD T0331  ; 进料移栽伸缩气缸伸出位延时
AND 1.08  ; 进料移栽料盘放料位有料感应（常闭）
LD W115.15  ; 进料旋转伺服在#1待料位
ANDNOT H51.05  ; 进料#1移栽位有料
ANDNOT H51.06  ; 进料#2移栽位有料
LD W116.00  ; 进料旋转伺服在#2待料位
ANDNOT H51.07  ; 进料#3移栽位有料
ANDNOT H51.08  ; 进料#4移栽位有料
ORLD
ANDLD
OR T0330  ; 进料旋转伸缩气缸缩回位延时
ANDLD
SET W110.09  ; 进料水平伺自动回服放料位辅助
; rung 42: 进料升降伺服回待料位
LD P_On
OUT TR0
AND 1401.07  ; 进料机构升降回待料位
TIMX(550) 0107 &3  ; 进料机构升降回待料位 延时
LD TR0
@LD 1401.03  ; 进料升降伺服取料后回待料位
@OR T0107  ; 进料机构升降回待料位 延时
@OR T0502  ; 自动回进料升降伺服待料位辅助延时
ANDLD
AND T0104  ; 进料升降伺服停止延时
AND W500.05  ; 升降触发条件
@SET W110.14  ; 自动回进料升降伺服待料位辅助

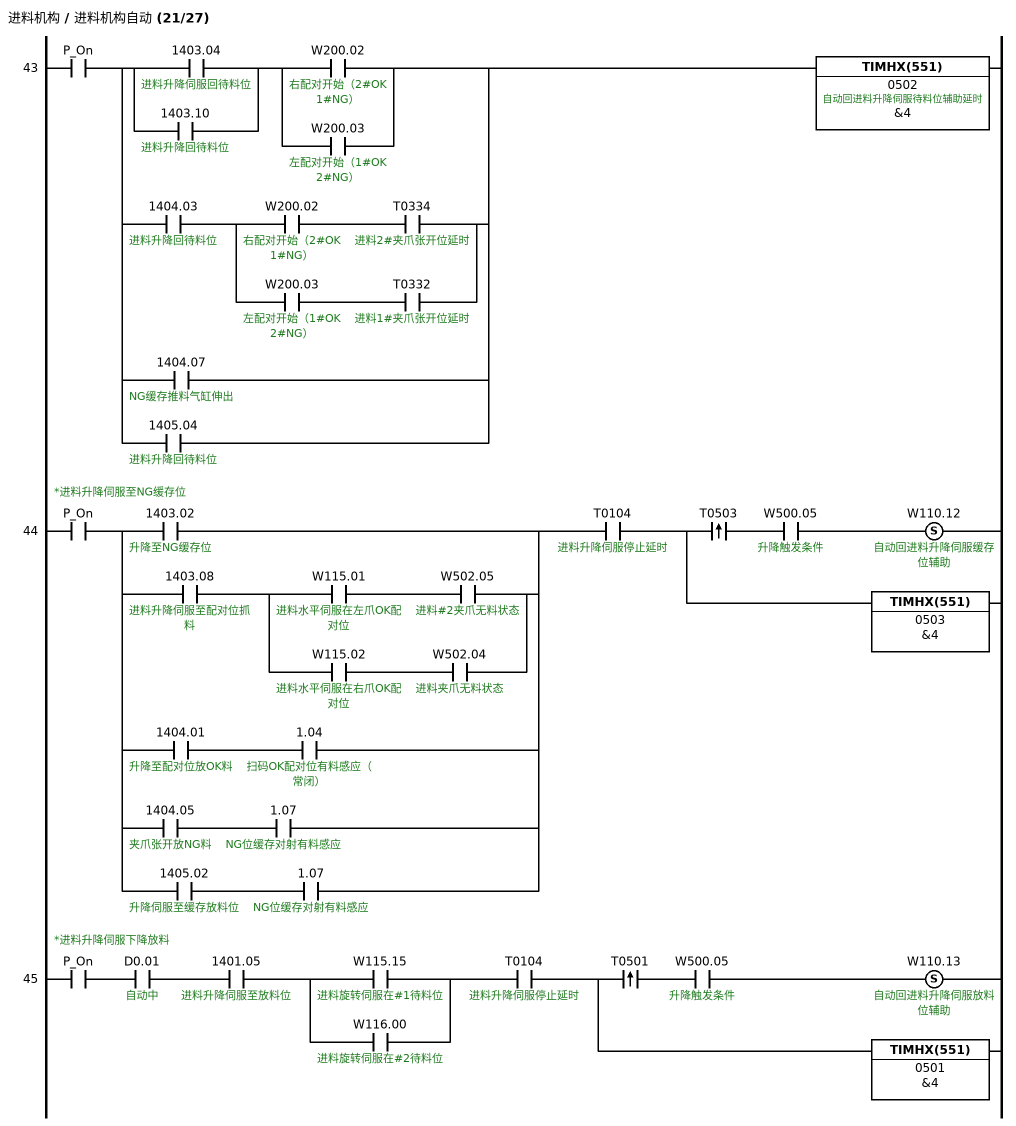
; rung 43
LD P_On
LD 1403.04  ; 进料升降伺服回待料位
OR 1403.10  ; 进料升降回待料位
LD W200.02  ; 右配对开始（2#OK 1#NG）
OR W200.03  ; 左配对开始（1#OK 2#NG）
ANDLD
LD 1404.03  ; 进料升降回待料位
LD W200.02  ; 右配对开始（2#OK 1#NG）
AND T0334  ; 进料2#夹爪张开位延时
LD W200.03  ; 左配对开始（1#OK 2#NG）
AND T0332  ; 进料1#夹爪张开位延时
ORLD
ANDLD
ORLD
OR 1404.07  ; NG缓存推料气缸伸出
OR 1405.04  ; 进料升降回待料位
ANDLD
TIMHX(551) 0502 &4  ; 自动回进料升降伺服待料位辅助延时
; rung 44: *进料升降伺服至NG缓存位
LD P_On
LD 1403.02  ; 升降至NG缓存位
LD 1403.08  ; 进料升降伺服至配对位抓料
LD W115.01  ; 进料水平伺服在左爪OK配对位
AND W502.05  ; 进料#2夹爪无料状态
LD W115.02  ; 进料水平伺服在右爪OK配对位
AND W502.04  ; 进料夹爪无料状态
ORLD
ANDLD
ORLD
LD 1404.01  ; 升降至配对位放OK料
AND 1.04  ; 扫码OK配对位有料感应（常闭）
ORLD
LD 1404.05  ; 夹爪张开放NG料
AND 1.07  ; NG位缓存对射有料感应
ORLD
LD 1405.02  ; 升降伺服至缓存放料位
AND 1.07  ; NG位缓存对射有料感应
ORLD
ANDLD
AND T0104  ; 进料升降伺服停止延时
OUT TR0
@AND T0503
AND W500.05  ; 升降触发条件
SET W110.12  ; 自动回进料升降伺服缓存位辅助
LD TR0
TIMHX(551) 0503 &4
; rung 45: *进料升降伺服下降放料
LD P_On
AND D0.01  ; 自动中
AND 1401.05  ; 进料升降伺服至放料位
LD W115.15  ; 进料旋转伺服在#1待料位
OR W116.00  ; 进料旋转伺服在#2待料位
ANDLD
AND T0104  ; 进料升降伺服停止延时
OUT TR0
@AND T0501
AND W500.05  ; 升降触发条件
SET W110.13  ; 自动回进料升降伺服放料位辅助
LD TR0
TIMHX(551) 0501 &4

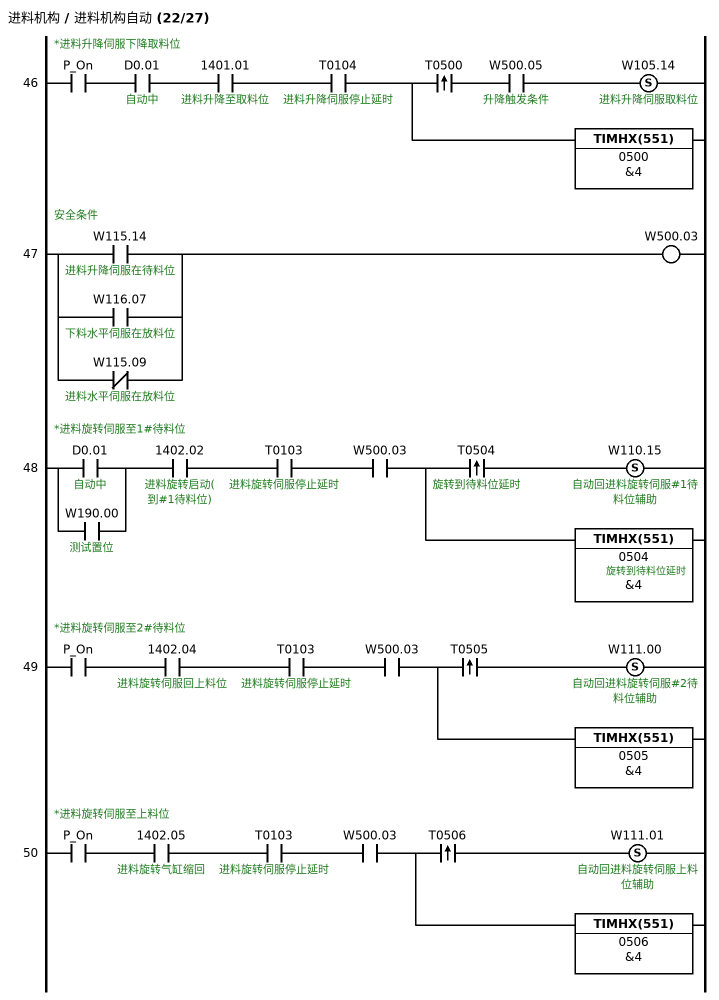
; rung 46: *进料升降伺服下降取料位
LD P_On
AND D0.01  ; 自动中
AND 1401.01  ; 进料升降至取料位
AND T0104  ; 进料升降伺服停止延时
OUT TR0
@AND T0500
AND W500.05  ; 升降触发条件
SET W105.14  ; 进料升降伺服取料位
LD TR0
TIMHX(551) 0500 &4
; rung 47: 安全条件
LD W115.14  ; 进料升降伺服在待料位
OR W116.07  ; 下料水平伺服在放料位
ORNOT W115.09  ; 进料水平伺服在放料位
OUT W500.03
; rung 48: *进料旋转伺服至1#待料位
LD D0.01  ; 自动中
OR W190.00  ; 测试置位
AND 1402.02  ; 进料旋转启动(到#1待料位)
AND T0103  ; 进料旋转伺服停止延时
AND W500.03
OUT TR0
@AND T0504  ; 旋转到待料位延时
SET W110.15  ; 自动回进料旋转伺服#1待料位辅助
LD TR0
TIMHX(551) 0504 &4  ; 旋转到待料位延时
; rung 49: *进料旋转伺服至2#待料位
LD P_On
AND 1402.04  ; 进料旋转伺服回上料位
AND T0103  ; 进料旋转伺服停止延时
AND W500.03
OUT TR0
@AND T0505
SET W111.00  ; 自动回进料旋转伺服#2待料位辅助
LD TR0
TIMHX(551) 0505 &4
; rung 50: *进料旋转伺服至上料位
LD P_On
AND 1402.05  ; 进料旋转气缸缩回
AND T0103  ; 进料旋转伺服停止延时
AND W500.03
OUT TR0
@AND T0506
SET W111.01  ; 自动回进料旋转伺服上料位辅助
LD TR0
TIMHX(551) 0506 &4

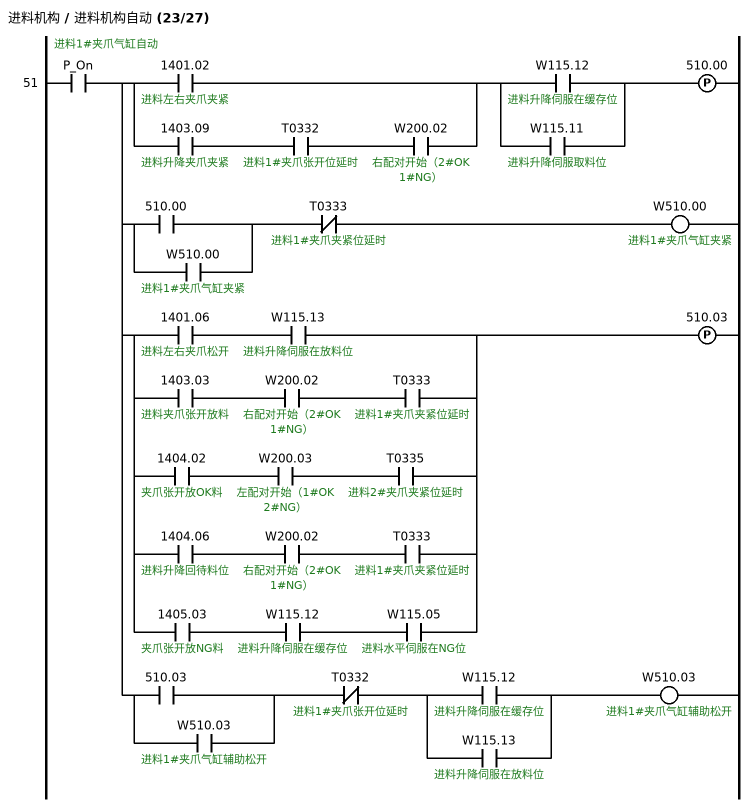
; rung 51: 进料1#夹爪气缸自动
LD P_On
OUT TR0
LD 1401.02  ; 进料左右夹爪夹紧
LD 1403.09  ; 进料升降夹爪夹紧
AND T0332  ; 进料1#夹爪张开位延时
AND W200.02  ; 右配对开始（2#OK 1#NG）
ORLD
ANDLD
LD W115.12  ; 进料升降伺服在缓存位
OR W115.11  ; 进料升降伺服取料位
ANDLD
DIFU(013) 510.00
LD TR0
LD 510.00
OR W510.00  ; 进料1#夹爪气缸夹紧
ANDLD
ANDNOT T0333  ; 进料1#夹爪夹紧位延时
OUT W510.00  ; 进料1#夹爪气缸夹紧
LD TR0
LD 1401.06  ; 进料左右夹爪松开
AND W115.13  ; 进料升降伺服在放料位
LD 1403.03  ; 进料夹爪张开放料
AND W200.02  ; 右配对开始（2#OK 1#NG）
AND T0333  ; 进料1#夹爪夹紧位延时
ORLD
LD 1404.02  ; 夹爪张开放OK料
AND W200.03  ; 左配对开始（1#OK 2#NG）
AND T0335  ; 进料2#夹爪夹紧位延时
ORLD
LD 1404.06  ; 进料升降回待料位
AND W200.02  ; 右配对开始（2#OK 1#NG）
AND T0333  ; 进料1#夹爪夹紧位延时
ORLD
LD 1405.03  ; 夹爪张开放NG料
AND W115.12  ; 进料升降伺服在缓存位
AND W115.05  ; 进料水平伺服在NG位
ORLD
ANDLD
DIFU(013) 510.03
LD TR0
LD 510.03
OR W510.03  ; 进料1#夹爪气缸辅助松开
ANDLD
ANDNOT T0332  ; 进料1#夹爪张开位延时
LD W115.12  ; 进料升降伺服在缓存位
OR W115.13  ; 进料升降伺服在放料位
ANDLD
OUT W510.03  ; 进料1#夹爪气缸辅助松开

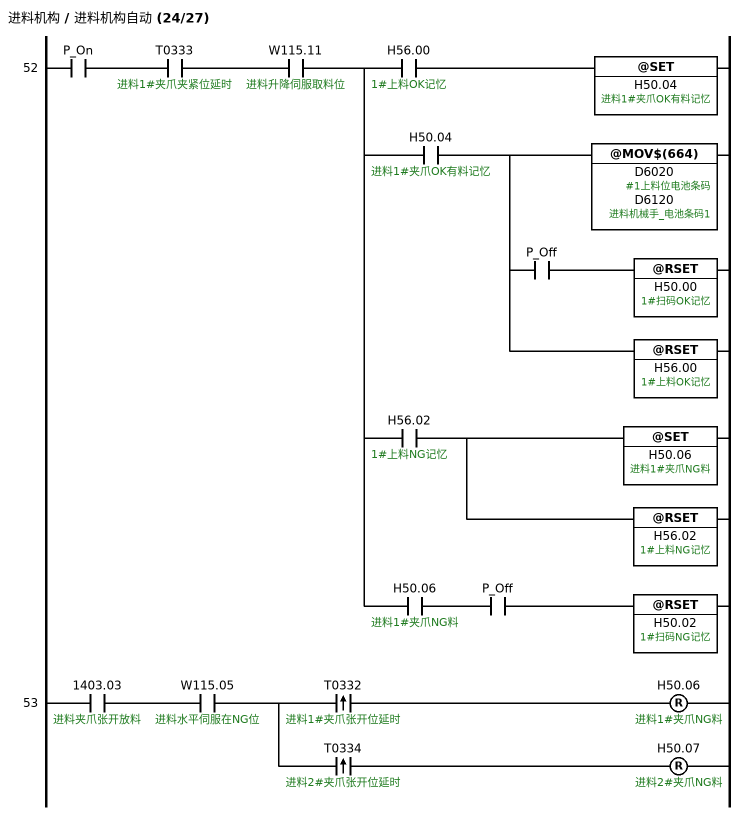
; rung 52
LD P_On
AND T0333  ; 进料1#夹爪夹紧位延时
AND W115.11  ; 进料升降伺服取料位
OUT TR0
AND H56.00  ; 1#上料OK记忆
@SET H50.04  ; 进料1#夹爪OK有料记忆
LD TR0
AND H50.04  ; 进料1#夹爪OK有料记忆
OUT TR1
@MOV$(664) D6020 D6120  ; #1上料位电池条码, 进料机械手_电池条码1
AND P_Off
@RSET H50.00  ; 1#扫码OK记忆
LD TR1
@RSET H56.00  ; 1#上料OK记忆
LD TR0
AND H56.02  ; 1#上料NG记忆
@SET H50.06  ; 进料1#夹爪NG料
@RSET H56.02  ; 1#上料NG记忆
LD TR0
AND H50.06  ; 进料1#夹爪NG料
AND P_Off
@RSET H50.02  ; 1#扫码NG记忆
; rung 53
LD 1403.03  ; 进料夹爪张开放料
AND W115.05  ; 进料水平伺服在NG位
OUT TR0
@AND T0332  ; 进料1#夹爪张开位延时
RSET H50.06  ; 进料1#夹爪NG料
LD TR0
@AND T0334  ; 进料2#夹爪张开位延时
RSET H50.07  ; 进料2#夹爪NG料

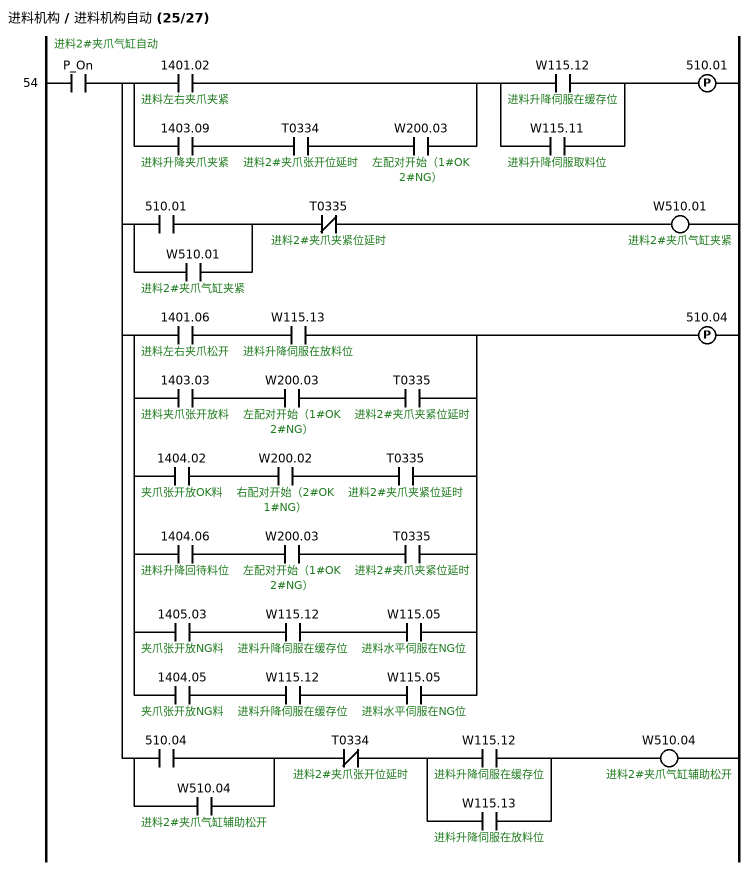
; rung 54: 进料2#夹爪气缸自动
LD P_On
OUT TR0
LD 1401.02  ; 进料左右夹爪夹紧
LD 1403.09  ; 进料升降夹爪夹紧
AND T0334  ; 进料2#夹爪张开位延时
AND W200.03  ; 左配对开始（1#OK 2#NG）
ORLD
ANDLD
LD W115.12  ; 进料升降伺服在缓存位
OR W115.11  ; 进料升降伺服取料位
ANDLD
DIFU(013) 510.01
LD TR0
LD 510.01
OR W510.01  ; 进料2#夹爪气缸夹紧
ANDLD
ANDNOT T0335  ; 进料2#夹爪夹紧位延时
OUT W510.01  ; 进料2#夹爪气缸夹紧
LD TR0
LD 1401.06  ; 进料左右夹爪松开
AND W115.13  ; 进料升降伺服在放料位
LD 1403.03  ; 进料夹爪张开放料
AND W200.03  ; 左配对开始（1#OK 2#NG）
AND T0335  ; 进料2#夹爪夹紧位延时
ORLD
LD 1404.02  ; 夹爪张开放OK料
AND W200.02  ; 右配对开始（2#OK 1#NG）
AND T0335  ; 进料2#夹爪夹紧位延时
ORLD
LD 1404.06  ; 进料升降回待料位
AND W200.03  ; 左配对开始（1#OK 2#NG）
AND T0335  ; 进料2#夹爪夹紧位延时
ORLD
LD 1405.03  ; 夹爪张开放NG料
AND W115.12  ; 进料升降伺服在缓存位
AND W115.05  ; 进料水平伺服在NG位
ORLD
LD 1404.05  ; 夹爪张开放NG料
AND W115.12  ; 进料升降伺服在缓存位
AND W115.05  ; 进料水平伺服在NG位
ORLD
ANDLD
DIFU(013) 510.04
LD TR0
LD 510.04
OR W510.04  ; 进料2#夹爪气缸辅助松开
ANDLD
ANDNOT T0334  ; 进料2#夹爪张开位延时
LD W115.12  ; 进料升降伺服在缓存位
OR W115.13  ; 进料升降伺服在放料位
ANDLD
OUT W510.04  ; 进料2#夹爪气缸辅助松开

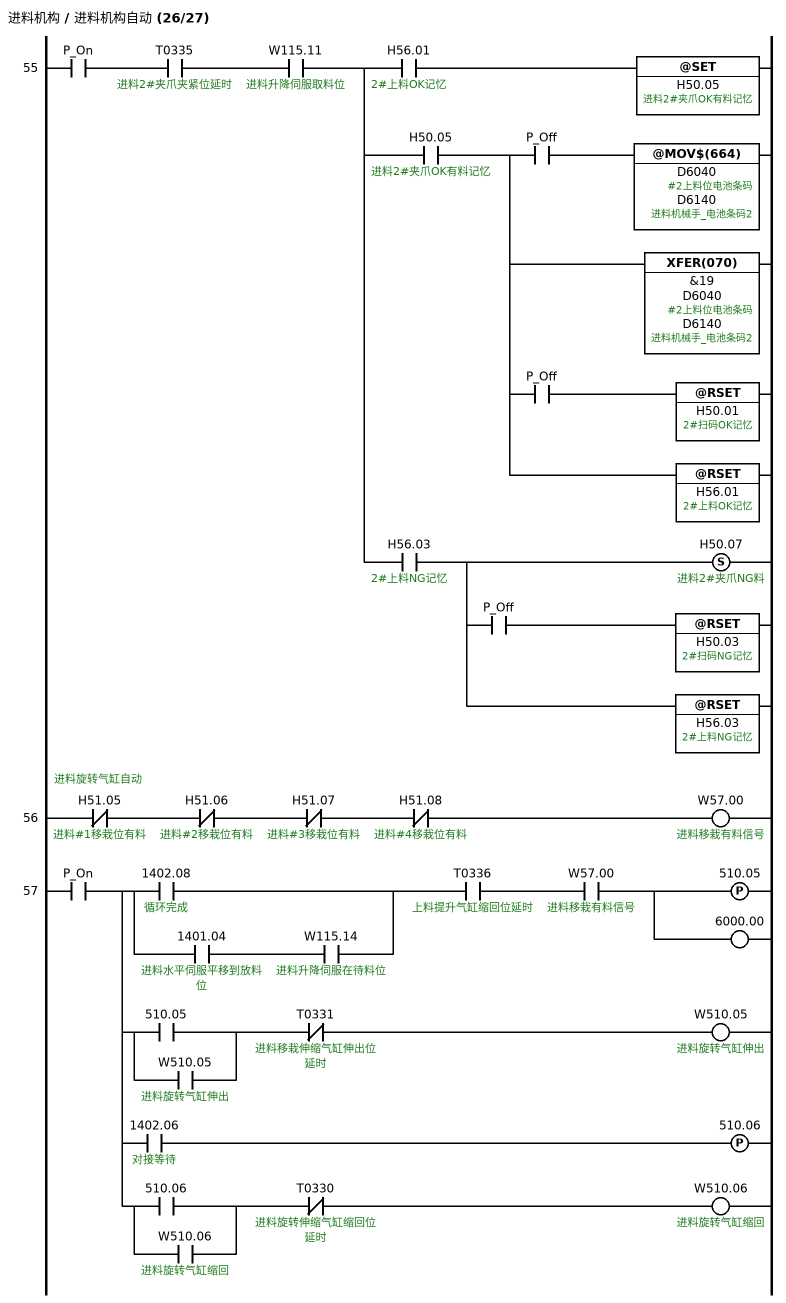
; rung 55
LD P_On
AND T0335  ; 进料2#夹爪夹紧位延时
AND W115.11  ; 进料升降伺服取料位
OUT TR0
AND H56.01  ; 2#上料OK记忆
@SET H50.05  ; 进料2#夹爪OK有料记忆
LD TR0
AND H50.05  ; 进料2#夹爪OK有料记忆
OUT TR1
AND P_Off
@MOV$(664) D6040 D6140  ; #2上料位电池条码, 进料机械手_电池条码2
LD TR1
XFER(070) &19 D6040 D6140  ; #2上料位电池条码, 进料机械手_电池条码2
AND P_Off
@RSET H50.01  ; 2#扫码OK记忆
LD TR1
@RSET H56.01  ; 2#上料OK记忆
LD TR0
AND H56.03  ; 2#上料NG记忆
OUT TR0
SET H50.07  ; 进料2#夹爪NG料
AND P_Off
@RSET H50.03  ; 2#扫码NG记忆
LD TR0
@RSET H56.03  ; 2#上料NG记忆
; rung 56: 进料旋转气缸自动
LDNOT H51.05  ; 进料#1移栽位有料
ANDNOT H51.06  ; 进料#2移栽位有料
ANDNOT H51.07  ; 进料#3移栽位有料
ANDNOT H51.08  ; 进料#4移栽位有料
OUT W57.00  ; 进料移栽有料信号
; rung 57
LD P_On
OUT TR0
LD 1402.08  ; 循环完成
LD 1401.04  ; 进料水平伺服平移到放料位
AND W115.14  ; 进料升降伺服在待料位
ORLD
ANDLD
AND T0336  ; 上料提升气缸缩回位延时
AND W57.00  ; 进料移栽有料信号
DIFU(013) 510.05
OUT 6000.00
LD TR0
LD 510.05
OR W510.05  ; 进料旋转气缸伸出
ANDLD
ANDNOT T0331  ; 进料移栽伸缩气缸伸出位延时
OUT W510.05  ; 进料旋转气缸伸出
LD TR0
AND 1402.06  ; 对接等待
DIFU(013) 510.06
LD TR0
LD 510.06
OR W510.06  ; 进料旋转气缸缩回
ANDLD
ANDNOT T0330  ; 进料旋转伸缩气缸缩回位延时
OUT W510.06  ; 进料旋转气缸缩回

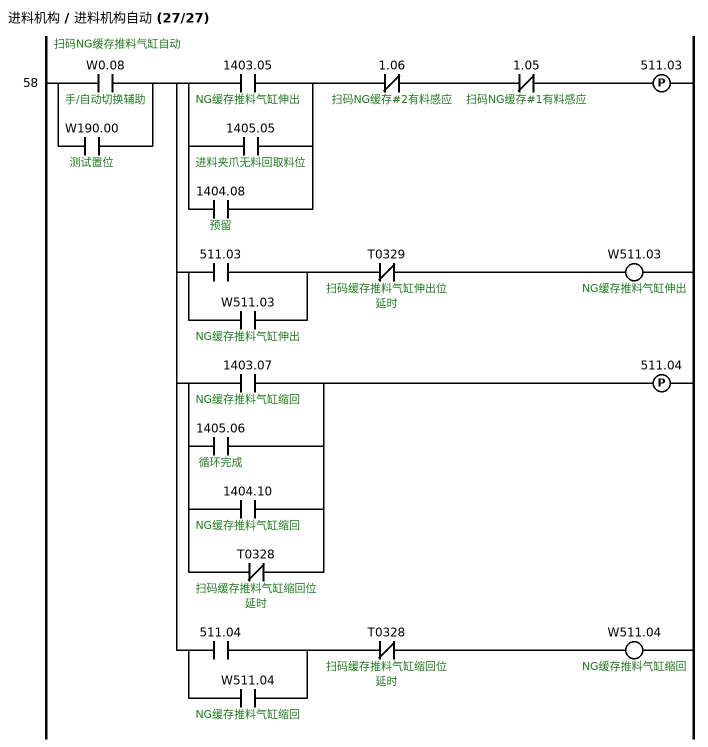
; rung 58: 扫码NG缓存推料气缸自动
LD W0.08  ; 手/自动切换辅助
OR W190.00  ; 测试置位
OUT TR0
LD 1403.05  ; NG缓存推料气缸伸出
OR 1405.05  ; 进料夹爪无料回取料位
OR 1404.08  ; 预留
ANDLD
ANDNOT 1.06  ; 扫码NG缓存#2有料感应
ANDNOT 1.05  ; 扫码NG缓存#1有料感应
DIFU(013) 511.03
LD TR0
LD 511.03
OR W511.03  ; NG缓存推料气缸伸出
ANDLD
ANDNOT T0329  ; 扫码缓存推料气缸伸出位延时
OUT W511.03  ; NG缓存推料气缸伸出
LD TR0
LD 1403.07  ; NG缓存推料气缸缩回
OR 1405.06  ; 循环完成
OR 1404.10  ; NG缓存推料气缸缩回
ORNOT T0328  ; 扫码缓存推料气缸缩回位延时
ANDLD
DIFU(013) 511.04
LD TR0
LD 511.04
OR W511.04  ; NG缓存推料气缸缩回
ANDLD
ANDNOT T0328  ; 扫码缓存推料气缸缩回位延时
OUT W511.04  ; NG缓存推料气缸缩回

### Section 进料机构手动

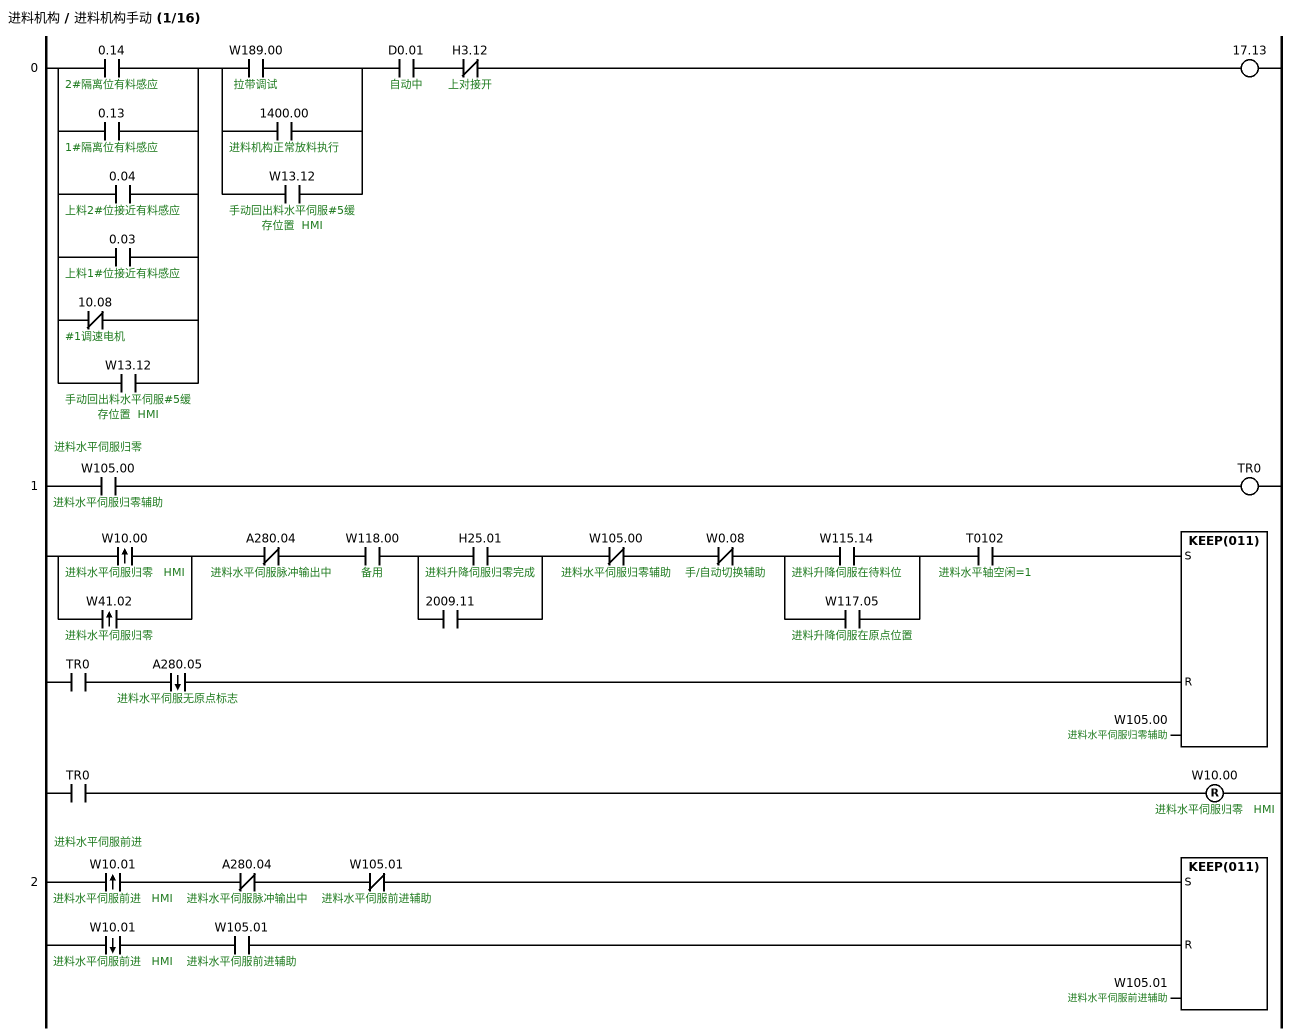
; rung 0
LD 0.14  ; 2#隔离位有料感应
OR 0.13  ; 1#隔离位有料感应
OR 0.04  ; 上料2#位接近有料感应
OR 0.03  ; 上料1#位接近有料感应
ORNOT 10.08  ; #1调速电机
OR W13.12  ; 手动回出料水平伺服#5缓存位置  HMI
LD W189.00  ; 拉带调试
OR 1400.00  ; 进料机构正常放料执行
OR W13.12  ; 手动回出料水平伺服#5缓存位置  HMI
ANDLD
AND D0.01  ; 自动中
ANDNOT H3.12  ; 上对接开
OUT 17.13
; rung 1: 进料水平伺服归零
@LD W10.00  ; 进料水平伺服归零   HMI
@OR W41.02  ; 进料水平伺服归零
ANDNOT A280.04  ; 进料水平伺服脉冲输出中
AND W118.00  ; 备用
LD H25.01  ; 进料升降伺服归零完成
OR 2009.11
ANDLD
ANDNOT W105.00  ; 进料水平伺服归零辅助
ANDNOT W0.08  ; 手/自动切换辅助
LD W115.14  ; 进料升降伺服在待料位
OR W117.05  ; 进料升降伺服在原点位置
ANDLD
AND T0102  ; 进料水平轴空闲=1
LD W105.00  ; 进料水平伺服归零辅助
OUT TR0
%AND A280.05  ; 进料水平伺服无原点标志
KEEP(011) W105.00  ; 进料水平伺服归零辅助
LD TR0
RSET W10.00  ; 进料水平伺服归零   HMI
; rung 2: 进料水平伺服前进
@LD W10.01  ; 进料水平伺服前进   HMI
ANDNOT A280.04  ; 进料水平伺服脉冲输出中
ANDNOT W105.01  ; 进料水平伺服前进辅助
%LD W10.01  ; 进料水平伺服前进   HMI
AND W105.01  ; 进料水平伺服前进辅助
KEEP(011) W105.01  ; 进料水平伺服前进辅助

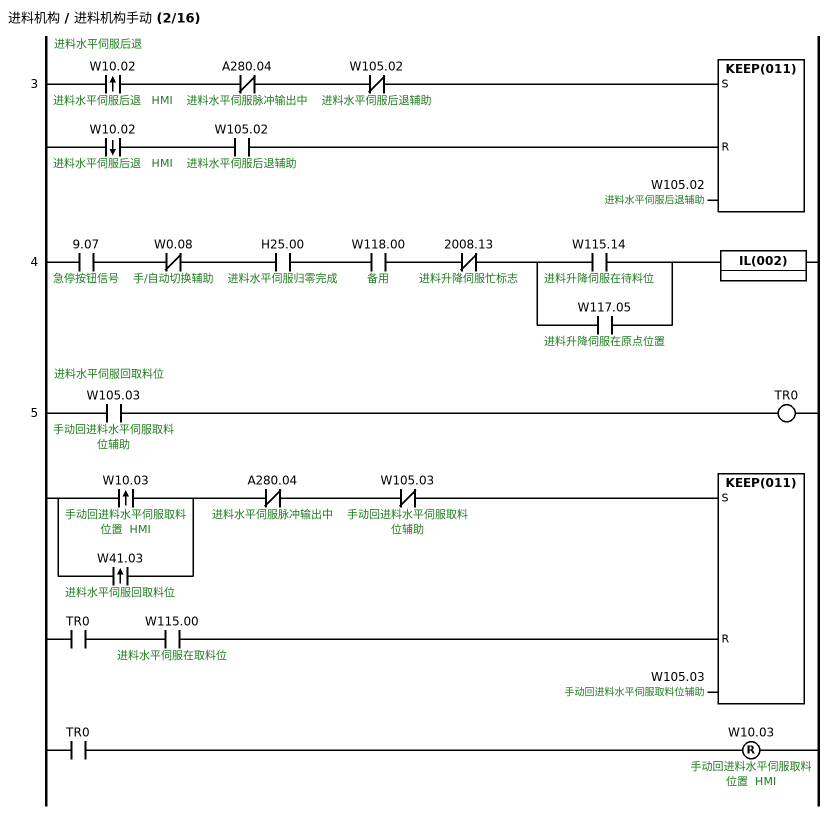
; rung 3: 进料水平伺服后退
@LD W10.02  ; 进料水平伺服后退   HMI
ANDNOT A280.04  ; 进料水平伺服脉冲输出中
ANDNOT W105.02  ; 进料水平伺服后退辅助
%LD W10.02  ; 进料水平伺服后退   HMI
AND W105.02  ; 进料水平伺服后退辅助
KEEP(011) W105.02  ; 进料水平伺服后退辅助
; rung 4
LD 9.07  ; 急停按钮信号
ANDNOT W0.08  ; 手/自动切换辅助
AND H25.00  ; 进料水平伺服归零完成
AND W118.00  ; 备用
ANDNOT 2008.13  ; 进料升降伺服忙标志
LD W115.14  ; 进料升降伺服在待料位
OR W117.05  ; 进料升降伺服在原点位置
ANDLD
IL(002)
; rung 5: 进料水平伺服回取料位
@LD W10.03  ; 手动回进料水平伺服取料位置  HMI
@OR W41.03  ; 进料水平伺服回取料位
ANDNOT A280.04  ; 进料水平伺服脉冲输出中
ANDNOT W105.03  ; 手动回进料水平伺服取料位辅助
LD W105.03  ; 手动回进料水平伺服取料位辅助
OUT TR0
AND W115.00  ; 进料水平伺服在取料位
KEEP(011) W105.03  ; 手动回进料水平伺服取料位辅助
LD TR0
RSET W10.03  ; 手动回进料水平伺服取料位置  HMI

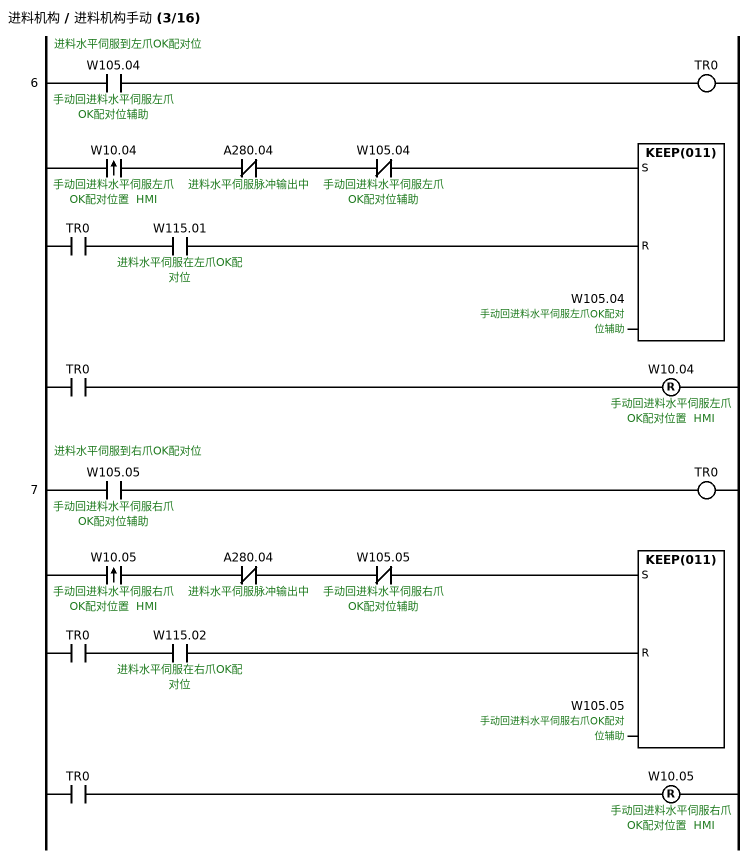
; rung 6: 进料水平伺服到左爪OK配对位
@LD W10.04  ; 手动回进料水平伺服左爪OK配对位置  HMI
ANDNOT A280.04  ; 进料水平伺服脉冲输出中
ANDNOT W105.04  ; 手动回进料水平伺服左爪OK配对位辅助
LD W105.04  ; 手动回进料水平伺服左爪OK配对位辅助
OUT TR0
AND W115.01  ; 进料水平伺服在左爪OK配对位
KEEP(011) W105.04  ; 手动回进料水平伺服左爪OK配对位辅助
LD TR0
RSET W10.04  ; 手动回进料水平伺服左爪OK配对位置  HMI
; rung 7: 进料水平伺服到右爪OK配对位
@LD W10.05  ; 手动回进料水平伺服右爪OK配对位置  HMI
ANDNOT A280.04  ; 进料水平伺服脉冲输出中
ANDNOT W105.05  ; 手动回进料水平伺服右爪OK配对位辅助
LD W105.05  ; 手动回进料水平伺服右爪OK配对位辅助
OUT TR0
AND W115.02  ; 进料水平伺服在右爪OK配对位
KEEP(011) W105.05  ; 手动回进料水平伺服右爪OK配对位辅助
LD TR0
RSET W10.05  ; 手动回进料水平伺服右爪OK配对位置  HMI

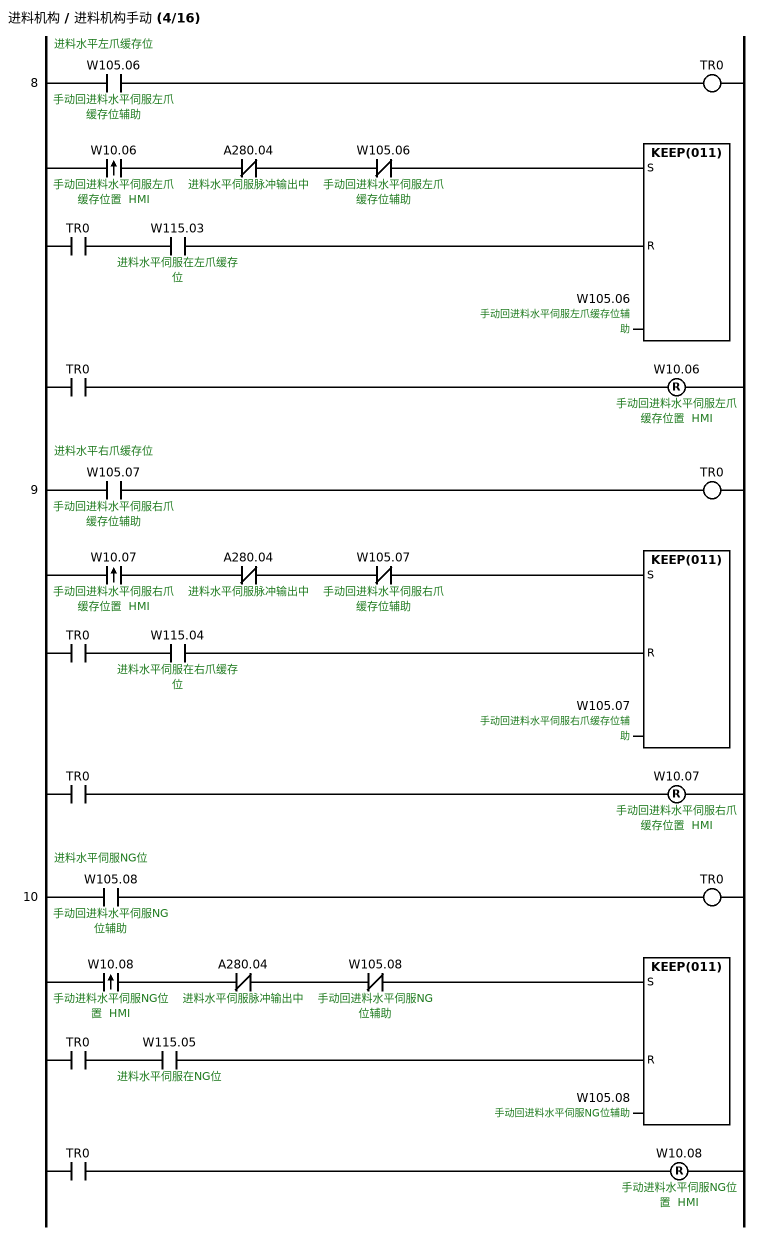
; rung 8: 进料水平左爪缓存位
@LD W10.06  ; 手动回进料水平伺服左爪缓存位置  HMI
ANDNOT A280.04  ; 进料水平伺服脉冲输出中
ANDNOT W105.06  ; 手动回进料水平伺服左爪缓存位辅助
LD W105.06  ; 手动回进料水平伺服左爪缓存位辅助
OUT TR0
AND W115.03  ; 进料水平伺服在左爪缓存位
KEEP(011) W105.06  ; 手动回进料水平伺服左爪缓存位辅助
LD TR0
RSET W10.06  ; 手动回进料水平伺服左爪缓存位置  HMI
; rung 9: 进料水平右爪缓存位
@LD W10.07  ; 手动回进料水平伺服右爪缓存位置  HMI
ANDNOT A280.04  ; 进料水平伺服脉冲输出中
ANDNOT W105.07  ; 手动回进料水平伺服右爪缓存位辅助
LD W105.07  ; 手动回进料水平伺服右爪缓存位辅助
OUT TR0
AND W115.04  ; 进料水平伺服在右爪缓存位
KEEP(011) W105.07  ; 手动回进料水平伺服右爪缓存位辅助
LD TR0
RSET W10.07  ; 手动回进料水平伺服右爪缓存位置  HMI
; rung 10: 进料水平伺服NG位
@LD W10.08  ; 手动进料水平伺服NG位置  HMI
ANDNOT A280.04  ; 进料水平伺服脉冲输出中
ANDNOT W105.08  ; 手动回进料水平伺服NG位辅助
LD W105.08  ; 手动回进料水平伺服NG位辅助
OUT TR0
AND W115.05  ; 进料水平伺服在NG位
KEEP(011) W105.08  ; 手动回进料水平伺服NG位辅助
LD TR0
RSET W10.08  ; 手动进料水平伺服NG位置  HMI

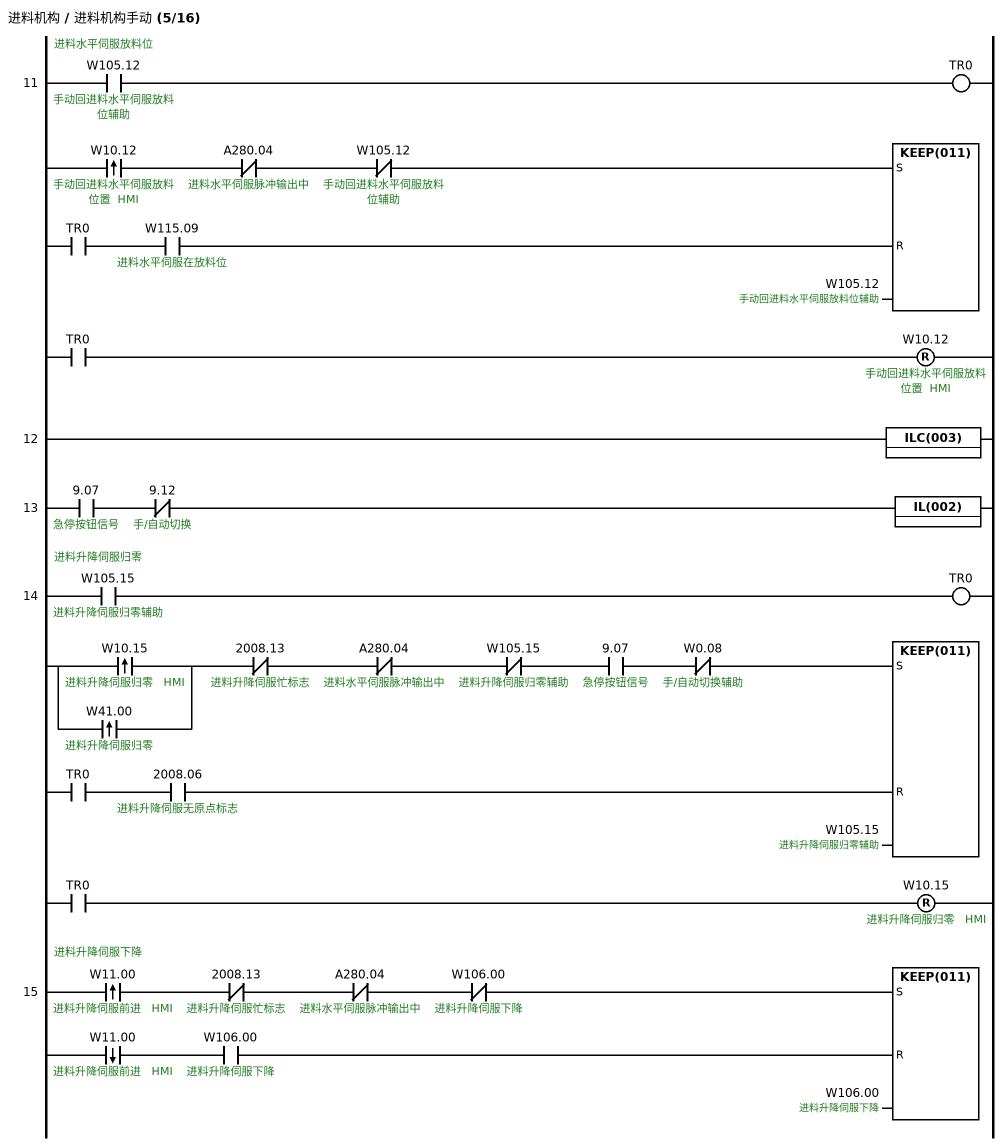
; rung 11: 进料水平伺服放料位
@LD W10.12  ; 手动回进料水平伺服放料位置  HMI
ANDNOT A280.04  ; 进料水平伺服脉冲输出中
ANDNOT W105.12  ; 手动回进料水平伺服放料位辅助
LD W105.12  ; 手动回进料水平伺服放料位辅助
OUT TR0
AND W115.09  ; 进料水平伺服在放料位
KEEP(011) W105.12  ; 手动回进料水平伺服放料位辅助
LD TR0
RSET W10.12  ; 手动回进料水平伺服放料位置  HMI
; rung 12
ILC(003)
; rung 13
LD 9.07  ; 急停按钮信号
ANDNOT 9.12  ; 手/自动切换
IL(002)
; rung 14: 进料升降伺服归零
@LD W10.15  ; 进料升降伺服归零   HMI
@OR W41.00  ; 进料升降伺服归零
ANDNOT 2008.13  ; 进料升降伺服忙标志
ANDNOT A280.04  ; 进料水平伺服脉冲输出中
ANDNOT W105.15  ; 进料升降伺服归零辅助
AND 9.07  ; 急停按钮信号
ANDNOT W0.08  ; 手/自动切换辅助
LD W105.15  ; 进料升降伺服归零辅助
OUT TR0
AND 2008.06  ; 进料升降伺服无原点标志
KEEP(011) W105.15  ; 进料升降伺服归零辅助
LD TR0
RSET W10.15  ; 进料升降伺服归零   HMI
; rung 15: 进料升降伺服下降
@LD W11.00  ; 进料升降伺服前进   HMI
ANDNOT 2008.13  ; 进料升降伺服忙标志
ANDNOT A280.04  ; 进料水平伺服脉冲输出中
ANDNOT W106.00  ; 进料升降伺服下降
%LD W11.00  ; 进料升降伺服前进   HMI
AND W106.00  ; 进料升降伺服下降
KEEP(011) W106.00  ; 进料升降伺服下降

